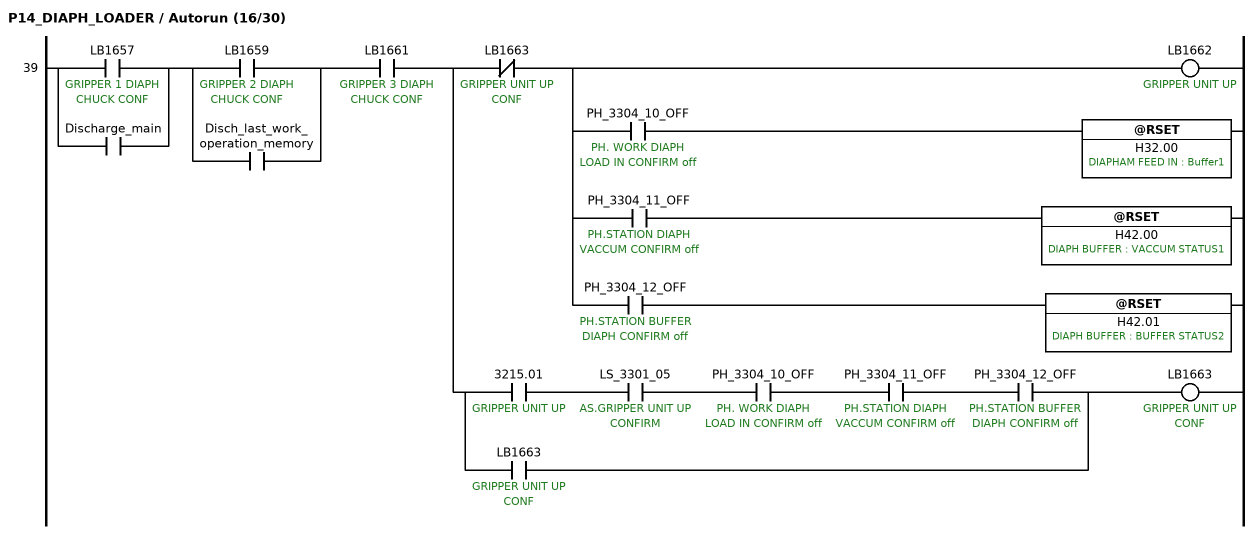
; [picture p192: P14_DIAPH_LOADER / Autorun, rungs 39-39]
; rung 39
LD LB1657  ; GRIPPER 1 DIAPH CHUCK CONF
OR Discharge_main
LD LB1659  ; GRIPPER 2 DIAPH CHUCK CONF
OR Disch_last_work_operation_memory
ANDLD
AND LB1661  ; GRIPPER 3 DIAPH CHUCK CONF
OUT TR0
ANDNOT LB1663  ; GRIPPER UNIT UP CONF
OUT TR1
OUT LB1662  ; GRIPPER UNIT UP
AND PH_3304_10_OFF  ; PH. WORK DIAPH LOAD IN CONFIRM off
@RSET H32.00  ; DIAPHAM FEED IN : Buffer1
LD TR1
AND PH_3304_11_OFF  ; PH.STATION DIAPH VACCUM CONFIRM off
@RSET H42.00  ; DIAPH BUFFER : VACCUM STATUS1
LD TR1
AND PH_3304_12_OFF  ; PH.STATION BUFFER DIAPH CONFIRM off
@RSET H42.01  ; DIAPH BUFFER : BUFFER STATUS2
LD TR0
LD 3215.01  ; GRIPPER UNIT UP
AND LS_3301_05  ; AS.GRIPPER UNIT UP CONFIRM
AND PH_3304_10_OFF  ; PH. WORK DIAPH LOAD IN CONFIRM off
AND PH_3304_11_OFF  ; PH.STATION DIAPH VACCUM CONFIRM off
AND PH_3304_12_OFF  ; PH.STATION BUFFER DIAPH CONFIRM off
OR LB1663  ; GRIPPER UNIT UP CONF
ANDLD
OUT LB1663  ; GRIPPER UNIT UP CONF

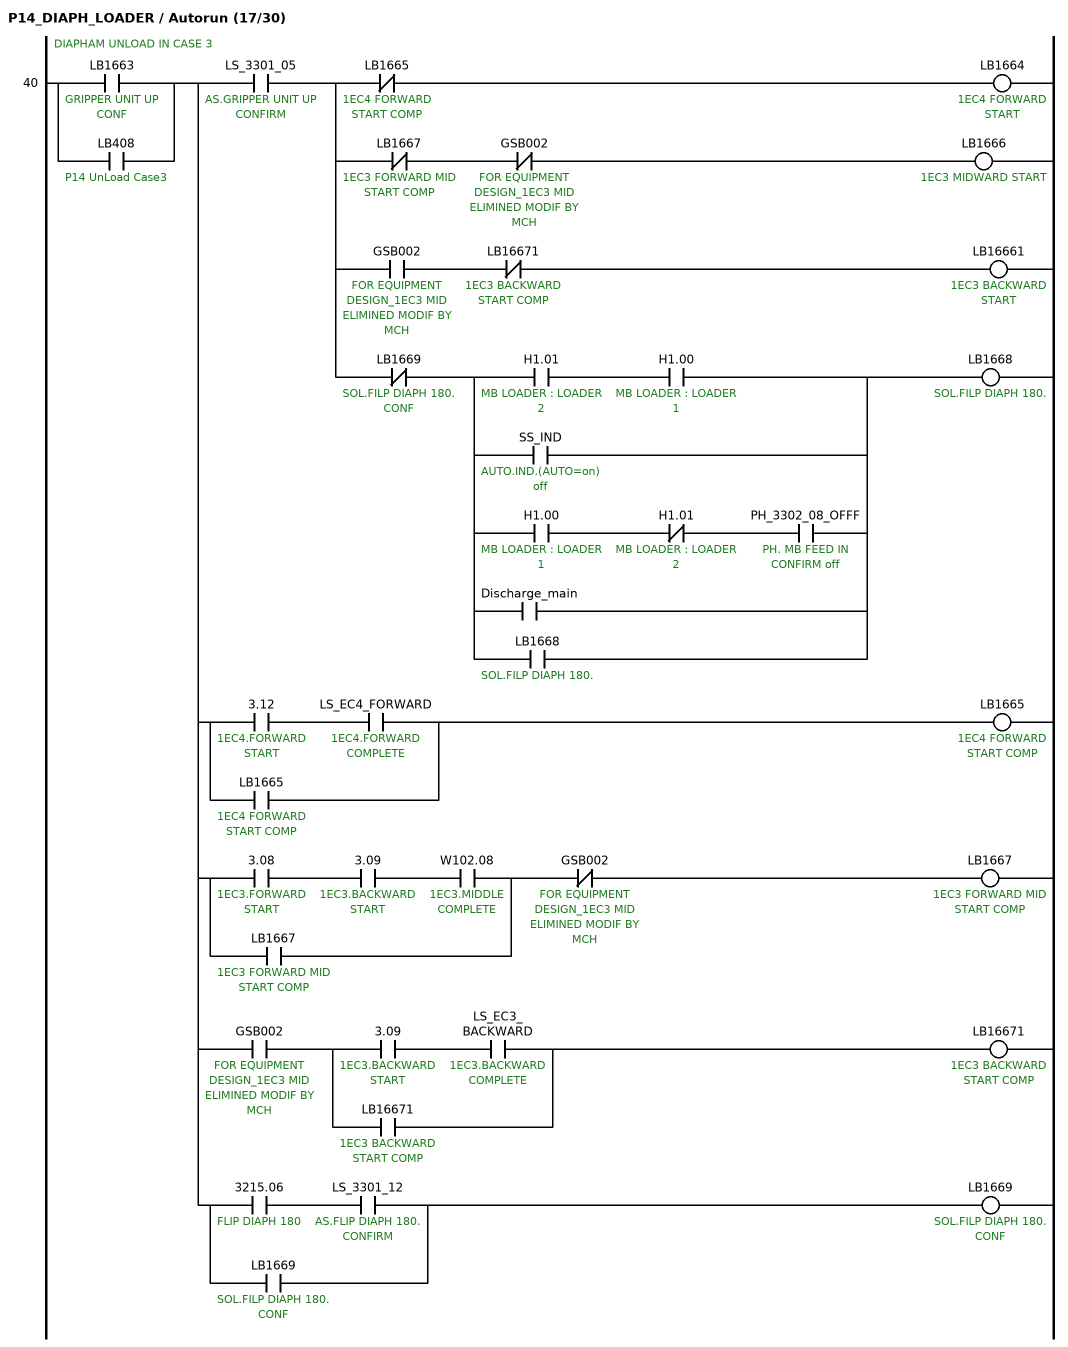
; rung 40: DIAPHAM UNLOAD IN CASE 3
LD LB1663  ; GRIPPER UNIT UP CONF
OR LB408  ; P14 UnLoad Case3
OUT TR0
AND LS_3301_05  ; AS.GRIPPER UNIT UP CONFIRM
OUT TR1
ANDNOT LB1665  ; 1EC4 FORWARD START COMP
OUT LB1664  ; 1EC4 FORWARD START
LD TR1
ANDNOT LB1667  ; 1EC3 FORWARD MID START COMP
ANDNOT GSB002  ; FOR EQUIPMENT DESIGN_1EC3 MID ELIMINED MODIF BY MCH
OUT LB1666  ; 1EC3 MIDWARD START
LD TR1
AND GSB002  ; FOR EQUIPMENT DESIGN_1EC3 MID ELIMINED MODIF BY MCH
ANDNOT LB16671  ; 1EC3 BACKWARD START COMP
OUT LB16661  ; 1EC3 BACKWARD START
LD TR1
ANDNOT LB1669  ; SOL.FILP DIAPH 180. CONF
LD H1.01  ; MB LOADER : LOADER 2
AND H1.00  ; MB LOADER : LOADER 1
OR SS_IND  ; AUTO.IND.(AUTO=on) off
LD H1.00  ; MB LOADER : LOADER 1
ANDNOT H1.01  ; MB LOADER : LOADER 2
AND PH_3302_08_OFFF  ; PH. MB FEED IN CONFIRM off
ORLD
OR Discharge_main
OR LB1668  ; SOL.FILP DIAPH 180.
ANDLD
OUT LB1668  ; SOL.FILP DIAPH 180.
LD TR0
LD 3.12  ; 1EC4.FORWARD START
AND LS_EC4_FORWARD  ; 1EC4.FORWARD COMPLETE
OR LB1665  ; 1EC4 FORWARD START COMP
ANDLD
OUT LB1665  ; 1EC4 FORWARD START COMP
LD TR0
LD 3.08  ; 1EC3.FORWARD START
AND 3.09  ; 1EC3.BACKWARD START
AND W102.08  ; 1EC3.MIDDLE COMPLETE
OR LB1667  ; 1EC3 FORWARD MID START COMP
ANDLD
ANDNOT GSB002  ; FOR EQUIPMENT DESIGN_1EC3 MID ELIMINED MODIF BY MCH
OUT LB1667  ; 1EC3 FORWARD MID START COMP
LD TR0
AND GSB002  ; FOR EQUIPMENT DESIGN_1EC3 MID ELIMINED MODIF BY MCH
LD 3.09  ; 1EC3.BACKWARD START
AND LS_EC3_BACKWARD  ; 1EC3.BACKWARD COMPLETE
OR LB16671  ; 1EC3 BACKWARD START COMP
ANDLD
OUT LB16671  ; 1EC3 BACKWARD START COMP
LD TR0
LD 3215.06  ; FLIP DIAPH 180
AND LS_3301_12  ; AS.FLIP DIAPH 180. CONFIRM
OR LB1669  ; SOL.FILP DIAPH 180. CONF
ANDLD
OUT LB1669  ; SOL.FILP DIAPH 180. CONF

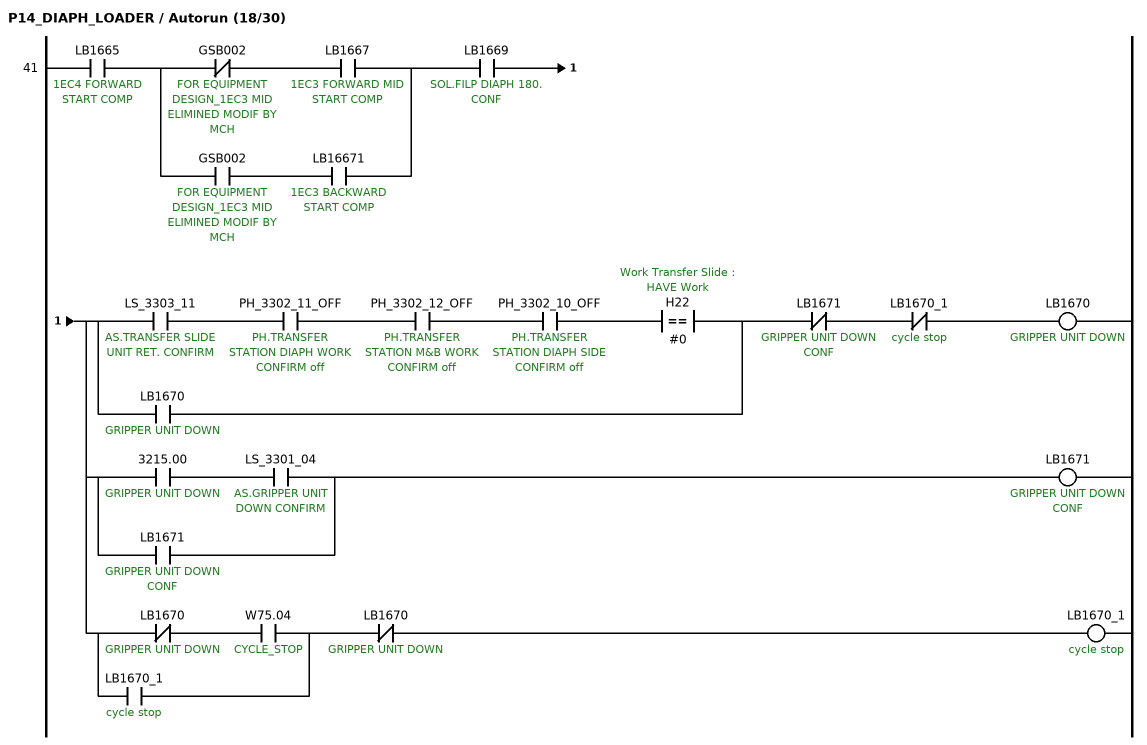
; rung 41
LD LB1665  ; 1EC4 FORWARD START COMP
LDNOT GSB002  ; FOR EQUIPMENT DESIGN_1EC3 MID ELIMINED MODIF BY MCH
AND LB1667  ; 1EC3 FORWARD MID START COMP
LD GSB002  ; FOR EQUIPMENT DESIGN_1EC3 MID ELIMINED MODIF BY MCH
AND LB16671  ; 1EC3 BACKWARD START COMP
ORLD
ANDLD
AND LB1669  ; SOL.FILP DIAPH 180. CONF
OUT TR0
LD LS_3303_11  ; AS.TRANSFER SLIDE UNIT RET. CONFIRM
AND PH_3302_11_OFF  ; PH.TRANSFER STATION DIAPH WORK CONFIRM off
AND PH_3302_12_OFF  ; PH.TRANSFER STATION M&B WORK CONFIRM off
AND PH_3302_10_OFF  ; PH.TRANSFER STATION DIAPH SIDE CONFIRM off
AND=(300) H22 #0  ; Work Transfer Slide : HAVE Work
OR LB1670  ; GRIPPER UNIT DOWN
ANDLD
ANDNOT LB1671  ; GRIPPER UNIT DOWN CONF
ANDNOT LB1670_1  ; cycle stop
OUT LB1670  ; GRIPPER UNIT DOWN
LD TR0
LD 3215.00  ; GRIPPER UNIT DOWN
AND LS_3301_04  ; AS.GRIPPER UNIT DOWN CONFIRM
OR LB1671  ; GRIPPER UNIT DOWN CONF
ANDLD
OUT LB1671  ; GRIPPER UNIT DOWN CONF
LD TR0
LDNOT LB1670  ; GRIPPER UNIT DOWN
AND W75.04  ; CYCLE_STOP
OR LB1670_1  ; cycle stop
ANDLD
ANDNOT LB1670  ; GRIPPER UNIT DOWN
OUT LB1670_1  ; cycle stop

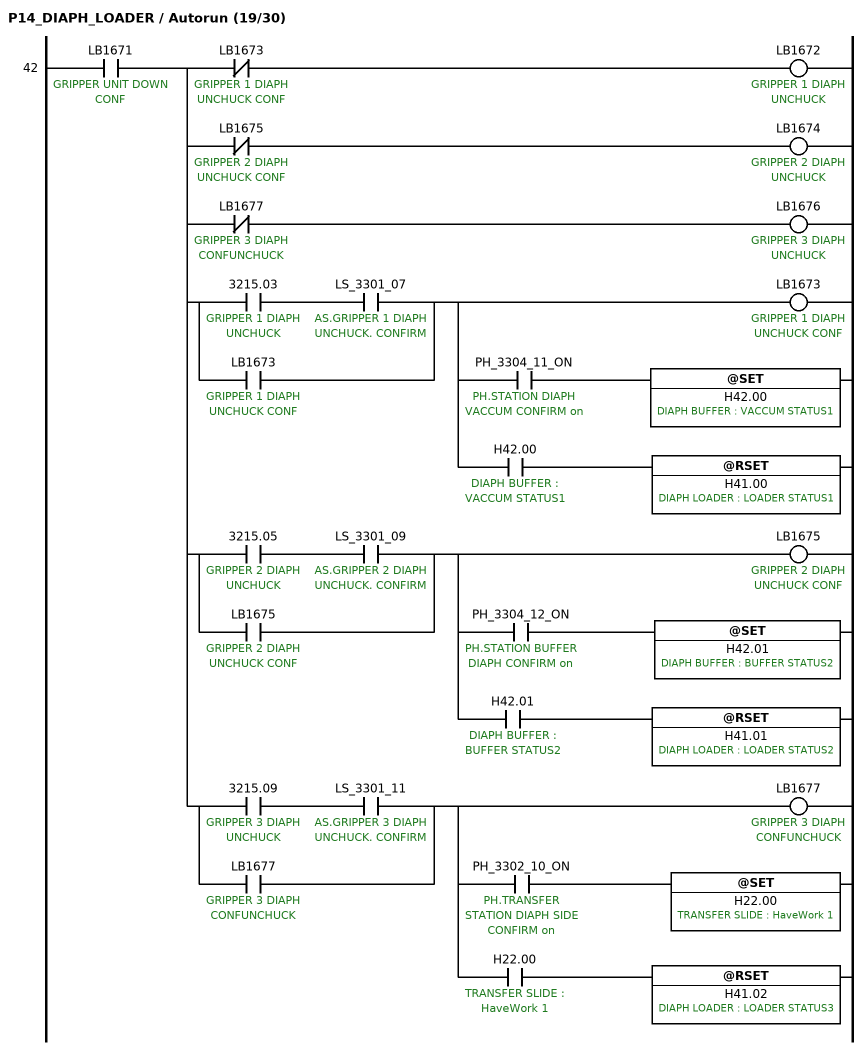
; rung 42
LD LB1671  ; GRIPPER UNIT DOWN CONF
OUT TR0
ANDNOT LB1673  ; GRIPPER 1 DIAPH UNCHUCK CONF
OUT LB1672  ; GRIPPER 1 DIAPH UNCHUCK
LD TR0
ANDNOT LB1675  ; GRIPPER 2 DIAPH UNCHUCK CONF
OUT LB1674  ; GRIPPER 2 DIAPH UNCHUCK
LD TR0
ANDNOT LB1677  ; GRIPPER 3 DIAPH CONFUNCHUCK
OUT LB1676  ; GRIPPER 3 DIAPH UNCHUCK
LD TR0
LD 3215.03  ; GRIPPER 1 DIAPH UNCHUCK
AND LS_3301_07  ; AS.GRIPPER 1 DIAPH UNCHUCK. CONFIRM
OR LB1673  ; GRIPPER 1 DIAPH UNCHUCK CONF
ANDLD
OUT TR1
OUT LB1673  ; GRIPPER 1 DIAPH UNCHUCK CONF
AND PH_3304_11_ON  ; PH.STATION DIAPH VACCUM CONFIRM on
@SET H42.00  ; DIAPH BUFFER : VACCUM STATUS1
LD TR1
AND H42.00  ; DIAPH BUFFER : VACCUM STATUS1
@RSET H41.00  ; DIAPH LOADER : LOADER STATUS1
LD TR0
LD 3215.05  ; GRIPPER 2 DIAPH UNCHUCK
AND LS_3301_09  ; AS.GRIPPER 2 DIAPH UNCHUCK. CONFIRM
OR LB1675  ; GRIPPER 2 DIAPH UNCHUCK CONF
ANDLD
OUT TR1
OUT LB1675  ; GRIPPER 2 DIAPH UNCHUCK CONF
AND PH_3304_12_ON  ; PH.STATION BUFFER DIAPH CONFIRM on
@SET H42.01  ; DIAPH BUFFER : BUFFER STATUS2
LD TR1
AND H42.01  ; DIAPH BUFFER : BUFFER STATUS2
@RSET H41.01  ; DIAPH LOADER : LOADER STATUS2
LD TR0
LD 3215.09  ; GRIPPER 3 DIAPH UNCHUCK
AND LS_3301_11  ; AS.GRIPPER 3 DIAPH UNCHUCK. CONFIRM
OR LB1677  ; GRIPPER 3 DIAPH CONFUNCHUCK
ANDLD
OUT TR0
OUT LB1677  ; GRIPPER 3 DIAPH CONFUNCHUCK
AND PH_3302_10_ON  ; PH.TRANSFER STATION DIAPH SIDE CONFIRM on
@SET H22.00  ; TRANSFER SLIDE : HaveWork 1
LD TR0
AND H22.00  ; TRANSFER SLIDE : HaveWork 1
@RSET H41.02  ; DIAPH LOADER : LOADER STATUS3

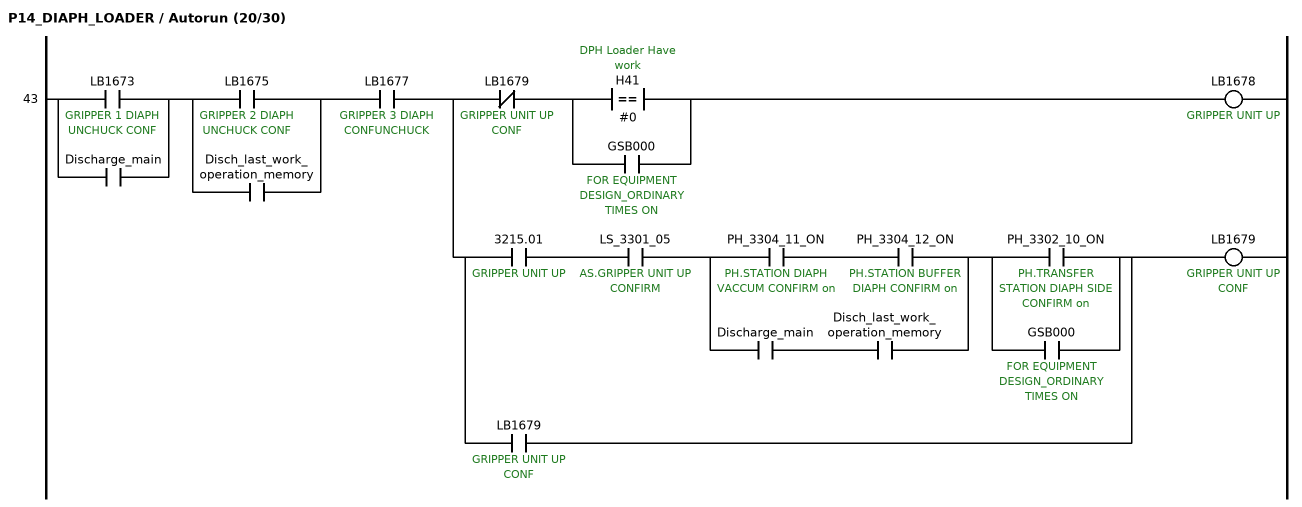
; rung 43
LD LB1673  ; GRIPPER 1 DIAPH UNCHUCK CONF
OR Discharge_main
LD LB1675  ; GRIPPER 2 DIAPH UNCHUCK CONF
OR Disch_last_work_operation_memory
ANDLD
AND LB1677  ; GRIPPER 3 DIAPH CONFUNCHUCK
OUT TR0
ANDNOT LB1679  ; GRIPPER UNIT UP CONF
LD=(300) H41 #0  ; DPH Loader Have work
OR GSB000  ; FOR EQUIPMENT DESIGN_ORDINARY TIMES ON
ANDLD
OUT LB1678  ; GRIPPER UNIT UP
LD TR0
LD 3215.01  ; GRIPPER UNIT UP
AND LS_3301_05  ; AS.GRIPPER UNIT UP CONFIRM
LD PH_3304_11_ON  ; PH.STATION DIAPH VACCUM CONFIRM on
AND PH_3304_12_ON  ; PH.STATION BUFFER DIAPH CONFIRM on
LD Discharge_main
AND Disch_last_work_operation_memory
ORLD
ANDLD
LD PH_3302_10_ON  ; PH.TRANSFER STATION DIAPH SIDE CONFIRM on
OR GSB000  ; FOR EQUIPMENT DESIGN_ORDINARY TIMES ON
ANDLD
OR LB1679  ; GRIPPER UNIT UP CONF
ANDLD
OUT LB1679  ; GRIPPER UNIT UP CONF

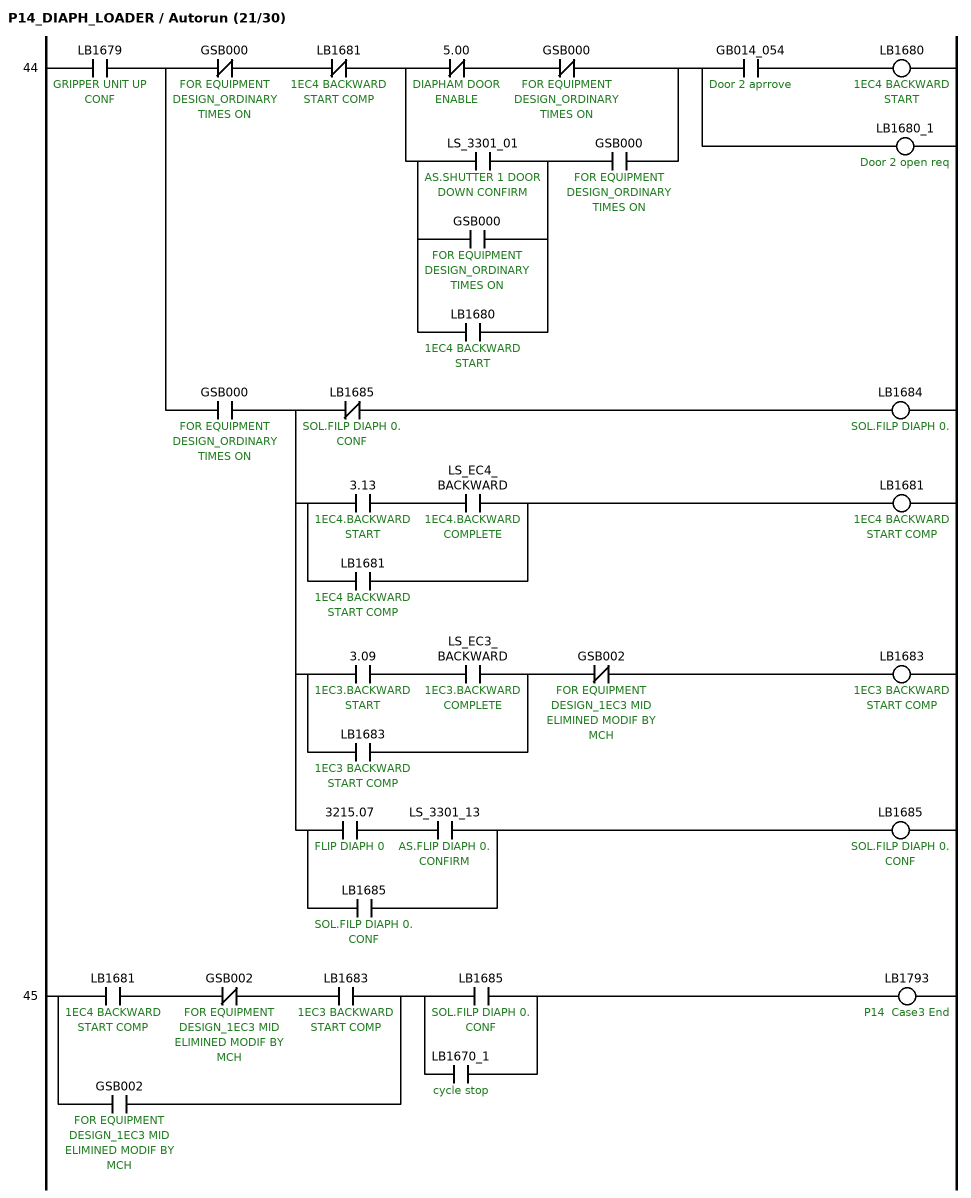
; rung 44
LD LB1679  ; GRIPPER UNIT UP CONF
OUT TR0
ANDNOT GSB000  ; FOR EQUIPMENT DESIGN_ORDINARY TIMES ON
ANDNOT LB1681  ; 1EC4 BACKWARD START COMP
LDNOT 5.00  ; DIAPHAM DOOR ENABLE
ANDNOT GSB000  ; FOR EQUIPMENT DESIGN_ORDINARY TIMES ON
LD LS_3301_01  ; AS.SHUTTER 1 DOOR DOWN CONFIRM
OR GSB000  ; FOR EQUIPMENT DESIGN_ORDINARY TIMES ON
OR LB1680  ; 1EC4 BACKWARD START
AND GSB000  ; FOR EQUIPMENT DESIGN_ORDINARY TIMES ON
ORLD
ANDLD
OUT TR1
AND GB014_054  ; Door 2 aprrove
OUT LB1680  ; 1EC4 BACKWARD START
LD TR1
OUT LB1680_1  ; Door 2 open req
LD TR0
AND GSB000  ; FOR EQUIPMENT DESIGN_ORDINARY TIMES ON
OUT TR0
ANDNOT LB1685  ; SOL.FILP DIAPH 0. CONF
OUT LB1684  ; SOL.FILP DIAPH 0.
LD TR0
LD 3.13  ; 1EC4.BACKWARD START
AND LS_EC4_BACKWARD  ; 1EC4.BACKWARD COMPLETE
OR LB1681  ; 1EC4 BACKWARD START COMP
ANDLD
OUT LB1681  ; 1EC4 BACKWARD START COMP
LD TR0
LD 3.09  ; 1EC3.BACKWARD START
AND LS_EC3_BACKWARD  ; 1EC3.BACKWARD COMPLETE
OR LB1683  ; 1EC3 BACKWARD START COMP
ANDLD
ANDNOT GSB002  ; FOR EQUIPMENT DESIGN_1EC3 MID ELIMINED MODIF BY MCH
OUT LB1683  ; 1EC3 BACKWARD START COMP
LD TR0
LD 3215.07  ; FLIP DIAPH 0
AND LS_3301_13  ; AS.FLIP DIAPH 0. CONFIRM
OR LB1685  ; SOL.FILP DIAPH 0. CONF
ANDLD
OUT LB1685  ; SOL.FILP DIAPH 0. CONF
; rung 45
LD LB1681  ; 1EC4 BACKWARD START COMP
ANDNOT GSB002  ; FOR EQUIPMENT DESIGN_1EC3 MID ELIMINED MODIF BY MCH
AND LB1683  ; 1EC3 BACKWARD START COMP
OR GSB002  ; FOR EQUIPMENT DESIGN_1EC3 MID ELIMINED MODIF BY MCH
LD LB1685  ; SOL.FILP DIAPH 0. CONF
OR LB1670_1  ; cycle stop
ANDLD
OUT LB1793  ; P14  Case3 End

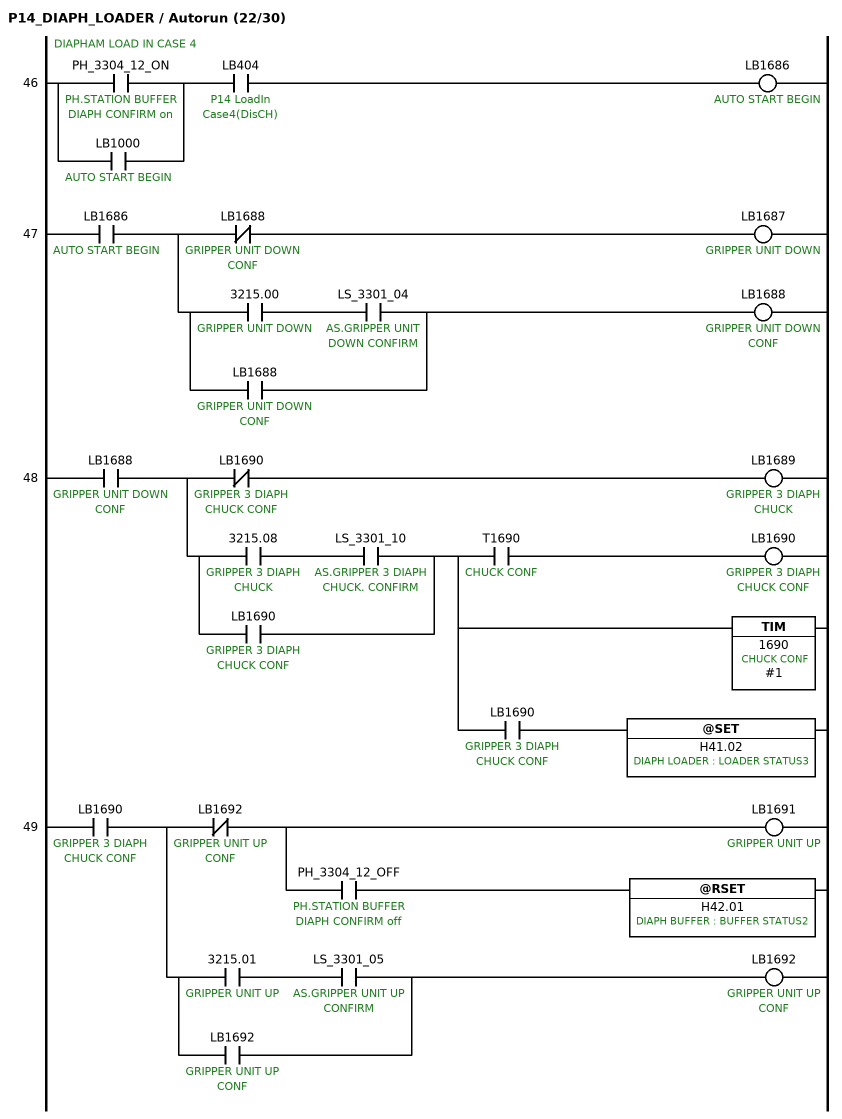
; rung 46: DIAPHAM LOAD IN CASE 4
LD PH_3304_12_ON  ; PH.STATION BUFFER DIAPH CONFIRM on
OR LB1000  ; AUTO START BEGIN
AND LB404  ; P14 LoadIn Case4(DisCH)
OUT LB1686  ; AUTO START BEGIN
; rung 47
LD LB1686  ; AUTO START BEGIN
OUT TR0
ANDNOT LB1688  ; GRIPPER UNIT DOWN CONF
OUT LB1687  ; GRIPPER UNIT DOWN
LD TR0
LD 3215.00  ; GRIPPER UNIT DOWN
AND LS_3301_04  ; AS.GRIPPER UNIT DOWN CONFIRM
OR LB1688  ; GRIPPER UNIT DOWN CONF
ANDLD
OUT LB1688  ; GRIPPER UNIT DOWN CONF
; rung 48
LD LB1688  ; GRIPPER UNIT DOWN CONF
OUT TR0
ANDNOT LB1690  ; GRIPPER 3 DIAPH CHUCK CONF
OUT LB1689  ; GRIPPER 3 DIAPH CHUCK
LD TR0
LD 3215.08  ; GRIPPER 3 DIAPH CHUCK
AND LS_3301_10  ; AS.GRIPPER 3 DIAPH CHUCK. CONFIRM
OR LB1690  ; GRIPPER 3 DIAPH CHUCK CONF
ANDLD
OUT TR0
AND T1690  ; CHUCK CONF
OUT LB1690  ; GRIPPER 3 DIAPH CHUCK CONF
LD TR0
TIM 1690 #1  ; CHUCK CONF
AND LB1690  ; GRIPPER 3 DIAPH CHUCK CONF
@SET H41.02  ; DIAPH LOADER : LOADER STATUS3
; rung 49
LD LB1690  ; GRIPPER 3 DIAPH CHUCK CONF
OUT TR0
ANDNOT LB1692  ; GRIPPER UNIT UP CONF
OUT LB1691  ; GRIPPER UNIT UP
AND PH_3304_12_OFF  ; PH.STATION BUFFER DIAPH CONFIRM off
@RSET H42.01  ; DIAPH BUFFER : BUFFER STATUS2
LD TR0
LD 3215.01  ; GRIPPER UNIT UP
AND LS_3301_05  ; AS.GRIPPER UNIT UP CONFIRM
OR LB1692  ; GRIPPER UNIT UP CONF
ANDLD
OUT LB1692  ; GRIPPER UNIT UP CONF

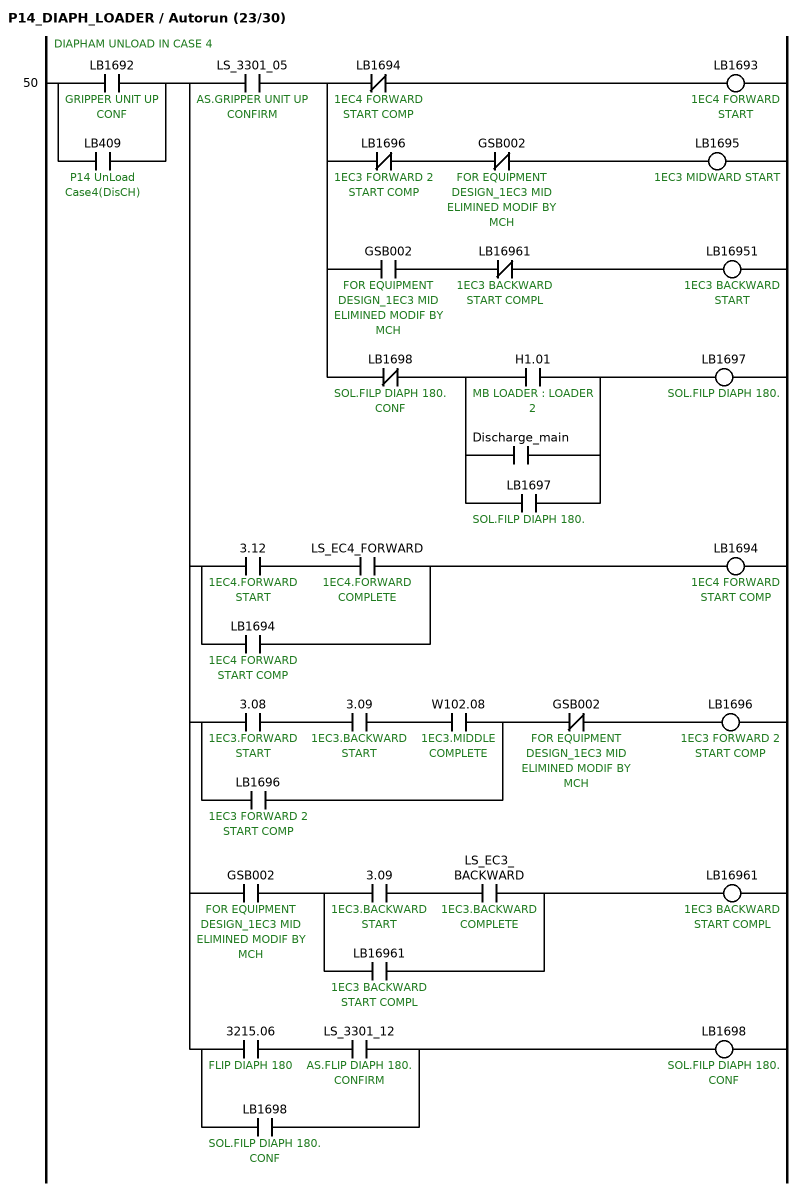
; rung 50: DIAPHAM UNLOAD IN CASE 4
LD LB1692  ; GRIPPER UNIT UP CONF
OR LB409  ; P14 UnLoad Case4(DisCH)
OUT TR0
AND LS_3301_05  ; AS.GRIPPER UNIT UP CONFIRM
OUT TR1
ANDNOT LB1694  ; 1EC4 FORWARD START COMP
OUT LB1693  ; 1EC4 FORWARD START
LD TR1
ANDNOT LB1696  ; 1EC3 FORWARD 2 START COMP
ANDNOT GSB002  ; FOR EQUIPMENT DESIGN_1EC3 MID ELIMINED MODIF BY MCH
OUT LB1695  ; 1EC3 MIDWARD START
LD TR1
AND GSB002  ; FOR EQUIPMENT DESIGN_1EC3 MID ELIMINED MODIF BY MCH
ANDNOT LB16961  ; 1EC3 BACKWARD START COMPL
OUT LB16951  ; 1EC3 BACKWARD START
LD TR1
ANDNOT LB1698  ; SOL.FILP DIAPH 180. CONF
LD H1.01  ; MB LOADER : LOADER 2
OR Discharge_main
OR LB1697  ; SOL.FILP DIAPH 180.
ANDLD
OUT LB1697  ; SOL.FILP DIAPH 180.
LD TR0
LD 3.12  ; 1EC4.FORWARD START
AND LS_EC4_FORWARD  ; 1EC4.FORWARD COMPLETE
OR LB1694  ; 1EC4 FORWARD START COMP
ANDLD
OUT LB1694  ; 1EC4 FORWARD START COMP
LD TR0
LD 3.08  ; 1EC3.FORWARD START
AND 3.09  ; 1EC3.BACKWARD START
AND W102.08  ; 1EC3.MIDDLE COMPLETE
OR LB1696  ; 1EC3 FORWARD 2 START COMP
ANDLD
ANDNOT GSB002  ; FOR EQUIPMENT DESIGN_1EC3 MID ELIMINED MODIF BY MCH
OUT LB1696  ; 1EC3 FORWARD 2 START COMP
LD TR0
AND GSB002  ; FOR EQUIPMENT DESIGN_1EC3 MID ELIMINED MODIF BY MCH
LD 3.09  ; 1EC3.BACKWARD START
AND LS_EC3_BACKWARD  ; 1EC3.BACKWARD COMPLETE
OR LB16961  ; 1EC3 BACKWARD START COMPL
ANDLD
OUT LB16961  ; 1EC3 BACKWARD START COMPL
LD TR0
LD 3215.06  ; FLIP DIAPH 180
AND LS_3301_12  ; AS.FLIP DIAPH 180. CONFIRM
OR LB1698  ; SOL.FILP DIAPH 180. CONF
ANDLD
OUT LB1698  ; SOL.FILP DIAPH 180. CONF

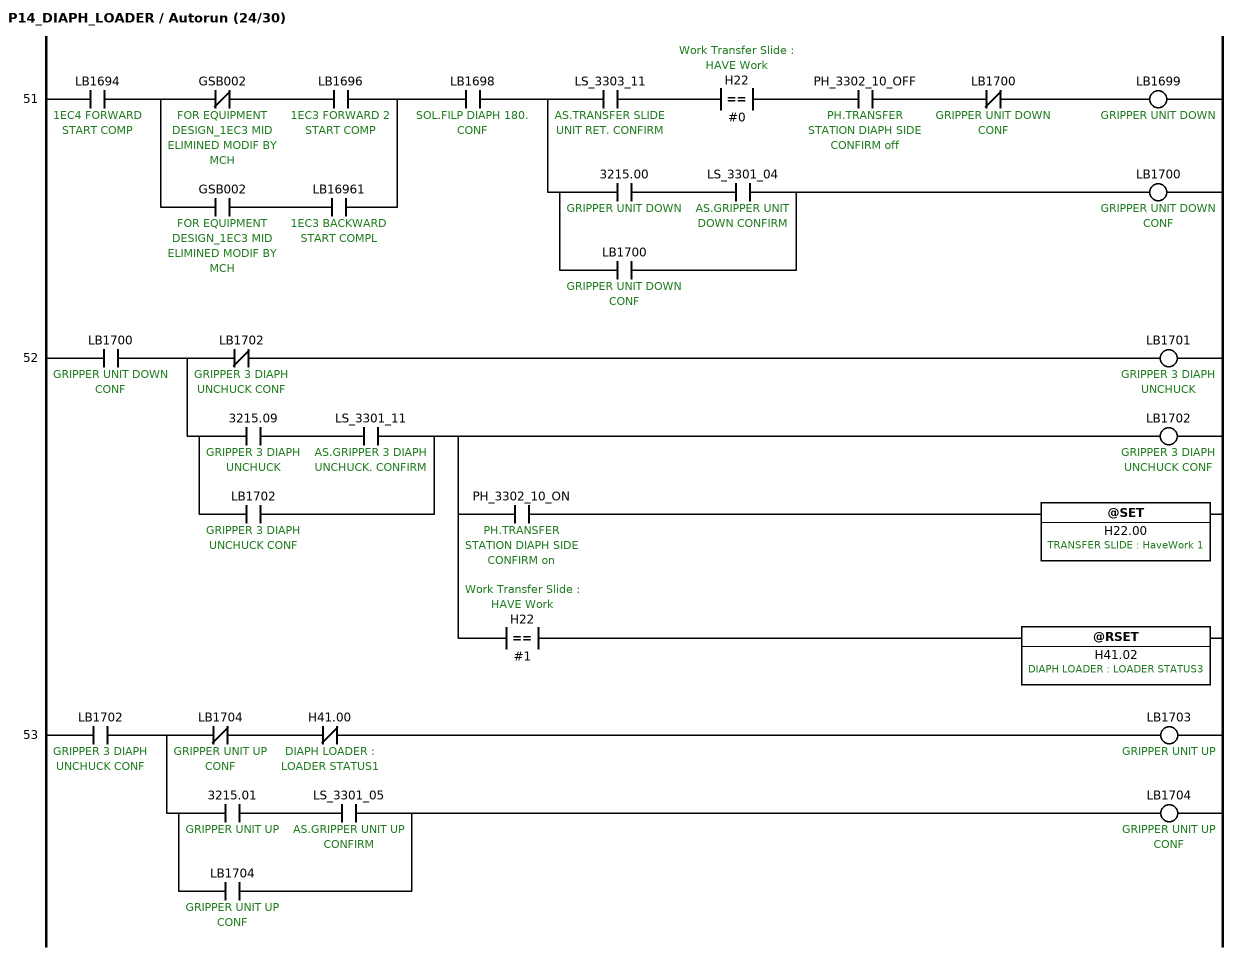
; rung 51
LD LB1694  ; 1EC4 FORWARD START COMP
LDNOT GSB002  ; FOR EQUIPMENT DESIGN_1EC3 MID ELIMINED MODIF BY MCH
AND LB1696  ; 1EC3 FORWARD 2 START COMP
LD GSB002  ; FOR EQUIPMENT DESIGN_1EC3 MID ELIMINED MODIF BY MCH
AND LB16961  ; 1EC3 BACKWARD START COMPL
ORLD
ANDLD
AND LB1698  ; SOL.FILP DIAPH 180. CONF
OUT TR0
AND LS_3303_11  ; AS.TRANSFER SLIDE UNIT RET. CONFIRM
AND=(300) H22 #0  ; Work Transfer Slide : HAVE Work
AND PH_3302_10_OFF  ; PH.TRANSFER STATION DIAPH SIDE CONFIRM off
ANDNOT LB1700  ; GRIPPER UNIT DOWN CONF
OUT LB1699  ; GRIPPER UNIT DOWN
LD TR0
LD 3215.00  ; GRIPPER UNIT DOWN
AND LS_3301_04  ; AS.GRIPPER UNIT DOWN CONFIRM
OR LB1700  ; GRIPPER UNIT DOWN CONF
ANDLD
OUT LB1700  ; GRIPPER UNIT DOWN CONF
; rung 52
LD LB1700  ; GRIPPER UNIT DOWN CONF
OUT TR0
ANDNOT LB1702  ; GRIPPER 3 DIAPH UNCHUCK CONF
OUT LB1701  ; GRIPPER 3 DIAPH UNCHUCK
LD TR0
LD 3215.09  ; GRIPPER 3 DIAPH UNCHUCK
AND LS_3301_11  ; AS.GRIPPER 3 DIAPH UNCHUCK. CONFIRM
OR LB1702  ; GRIPPER 3 DIAPH UNCHUCK CONF
ANDLD
OUT TR0
OUT LB1702  ; GRIPPER 3 DIAPH UNCHUCK CONF
AND PH_3302_10_ON  ; PH.TRANSFER STATION DIAPH SIDE CONFIRM on
@SET H22.00  ; TRANSFER SLIDE : HaveWork 1
LD TR0
AND=(300) H22 #1  ; Work Transfer Slide : HAVE Work
@RSET H41.02  ; DIAPH LOADER : LOADER STATUS3
; rung 53
LD LB1702  ; GRIPPER 3 DIAPH UNCHUCK CONF
OUT TR0
ANDNOT LB1704  ; GRIPPER UNIT UP CONF
ANDNOT H41.00  ; DIAPH LOADER : LOADER STATUS1
OUT LB1703  ; GRIPPER UNIT UP
LD TR0
LD 3215.01  ; GRIPPER UNIT UP
AND LS_3301_05  ; AS.GRIPPER UNIT UP CONFIRM
OR LB1704  ; GRIPPER UNIT UP CONF
ANDLD
OUT LB1704  ; GRIPPER UNIT UP CONF

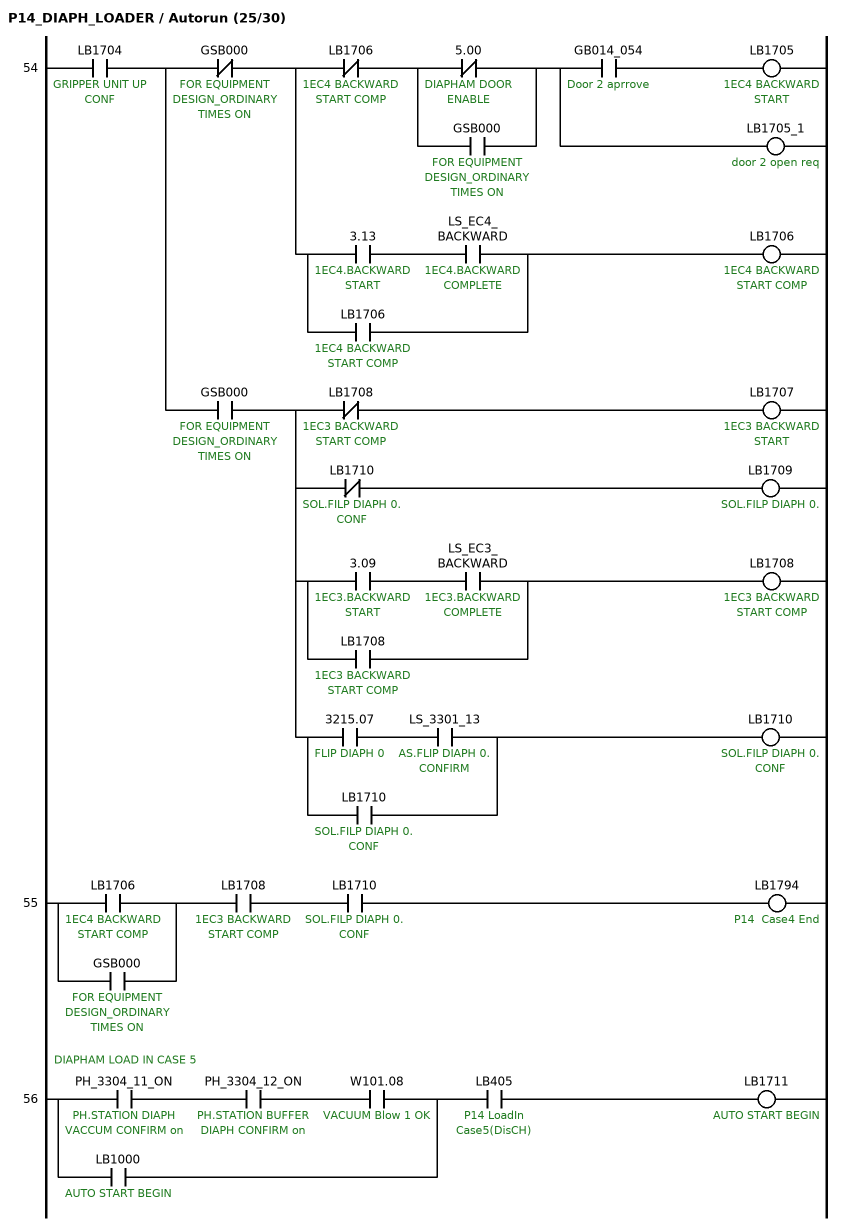
; rung 54
LD LB1704  ; GRIPPER UNIT UP CONF
OUT TR0
ANDNOT GSB000  ; FOR EQUIPMENT DESIGN_ORDINARY TIMES ON
OUT TR1
ANDNOT LB1706  ; 1EC4 BACKWARD START COMP
LDNOT 5.00  ; DIAPHAM DOOR ENABLE
OR GSB000  ; FOR EQUIPMENT DESIGN_ORDINARY TIMES ON
ANDLD
OUT TR2
AND GB014_054  ; Door 2 aprrove
OUT LB1705  ; 1EC4 BACKWARD START
LD TR2
OUT LB1705_1  ; door 2 open req
LD TR1
LD 3.13  ; 1EC4.BACKWARD START
AND LS_EC4_BACKWARD  ; 1EC4.BACKWARD COMPLETE
OR LB1706  ; 1EC4 BACKWARD START COMP
ANDLD
OUT LB1706  ; 1EC4 BACKWARD START COMP
LD TR0
AND GSB000  ; FOR EQUIPMENT DESIGN_ORDINARY TIMES ON
OUT TR0
ANDNOT LB1708  ; 1EC3 BACKWARD START COMP
OUT LB1707  ; 1EC3 BACKWARD START
LD TR0
ANDNOT LB1710  ; SOL.FILP DIAPH 0. CONF
OUT LB1709  ; SOL.FILP DIAPH 0.
LD TR0
LD 3.09  ; 1EC3.BACKWARD START
AND LS_EC3_BACKWARD  ; 1EC3.BACKWARD COMPLETE
OR LB1708  ; 1EC3 BACKWARD START COMP
ANDLD
OUT LB1708  ; 1EC3 BACKWARD START COMP
LD TR0
LD 3215.07  ; FLIP DIAPH 0
AND LS_3301_13  ; AS.FLIP DIAPH 0. CONFIRM
OR LB1710  ; SOL.FILP DIAPH 0. CONF
ANDLD
OUT LB1710  ; SOL.FILP DIAPH 0. CONF
; rung 55
LD LB1706  ; 1EC4 BACKWARD START COMP
OR GSB000  ; FOR EQUIPMENT DESIGN_ORDINARY TIMES ON
AND LB1708  ; 1EC3 BACKWARD START COMP
AND LB1710  ; SOL.FILP DIAPH 0. CONF
OUT LB1794  ; P14  Case4 End
; rung 56: DIAPHAM LOAD IN CASE 5
LD PH_3304_11_ON  ; PH.STATION DIAPH VACCUM CONFIRM on
AND PH_3304_12_ON  ; PH.STATION BUFFER DIAPH CONFIRM on
AND W101.08  ; VACUUM Blow 1 OK
OR LB1000  ; AUTO START BEGIN
AND LB405  ; P14 LoadIn Case5(DisCH)
OUT LB1711  ; AUTO START BEGIN

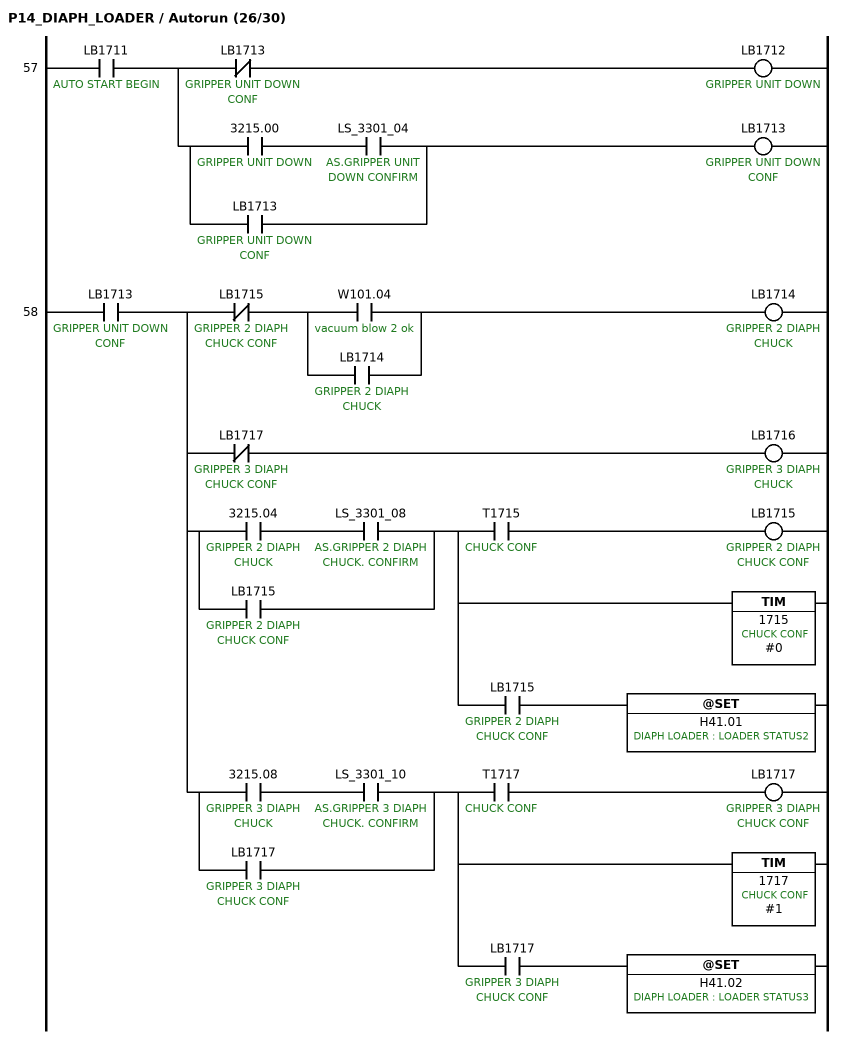
; rung 57
LD LB1711  ; AUTO START BEGIN
OUT TR0
ANDNOT LB1713  ; GRIPPER UNIT DOWN CONF
OUT LB1712  ; GRIPPER UNIT DOWN
LD TR0
LD 3215.00  ; GRIPPER UNIT DOWN
AND LS_3301_04  ; AS.GRIPPER UNIT DOWN CONFIRM
OR LB1713  ; GRIPPER UNIT DOWN CONF
ANDLD
OUT LB1713  ; GRIPPER UNIT DOWN CONF
; rung 58
LD LB1713  ; GRIPPER UNIT DOWN CONF
OUT TR0
ANDNOT LB1715  ; GRIPPER 2 DIAPH CHUCK CONF
LD W101.04  ; vacuum blow 2 ok
OR LB1714  ; GRIPPER 2 DIAPH CHUCK
ANDLD
OUT LB1714  ; GRIPPER 2 DIAPH CHUCK
LD TR0
ANDNOT LB1717  ; GRIPPER 3 DIAPH CHUCK CONF
OUT LB1716  ; GRIPPER 3 DIAPH CHUCK
LD TR0
LD 3215.04  ; GRIPPER 2 DIAPH CHUCK
AND LS_3301_08  ; AS.GRIPPER 2 DIAPH CHUCK. CONFIRM
OR LB1715  ; GRIPPER 2 DIAPH CHUCK CONF
ANDLD
OUT TR1
AND T1715  ; CHUCK CONF
OUT LB1715  ; GRIPPER 2 DIAPH CHUCK CONF
LD TR1
TIM 1715 #0  ; CHUCK CONF
AND LB1715  ; GRIPPER 2 DIAPH CHUCK CONF
@SET H41.01  ; DIAPH LOADER : LOADER STATUS2
LD TR0
LD 3215.08  ; GRIPPER 3 DIAPH CHUCK
AND LS_3301_10  ; AS.GRIPPER 3 DIAPH CHUCK. CONFIRM
OR LB1717  ; GRIPPER 3 DIAPH CHUCK CONF
ANDLD
OUT TR0
AND T1717  ; CHUCK CONF
OUT LB1717  ; GRIPPER 3 DIAPH CHUCK CONF
LD TR0
TIM 1717 #1  ; CHUCK CONF
AND LB1717  ; GRIPPER 3 DIAPH CHUCK CONF
@SET H41.02  ; DIAPH LOADER : LOADER STATUS3

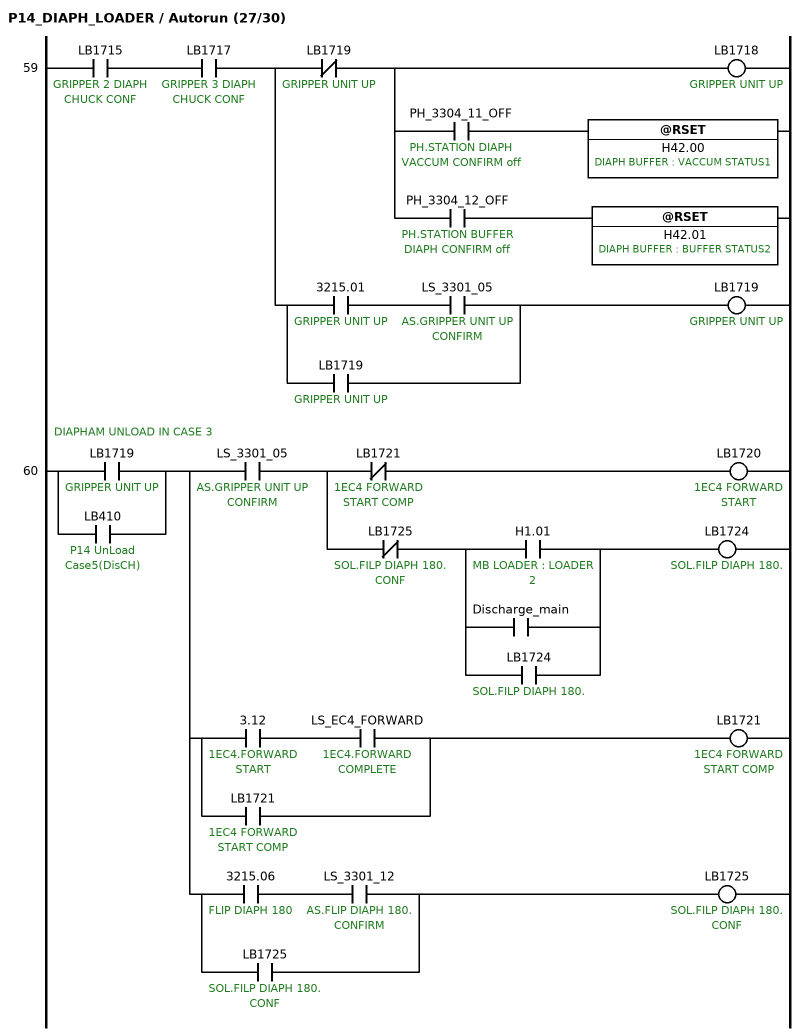
; rung 59
LD LB1715  ; GRIPPER 2 DIAPH CHUCK CONF
AND LB1717  ; GRIPPER 3 DIAPH CHUCK CONF
OUT TR0
ANDNOT LB1719  ; GRIPPER UNIT UP
OUT TR1
OUT LB1718  ; GRIPPER UNIT UP
AND PH_3304_11_OFF  ; PH.STATION DIAPH VACCUM CONFIRM off
@RSET H42.00  ; DIAPH BUFFER : VACCUM STATUS1
LD TR1
AND PH_3304_12_OFF  ; PH.STATION BUFFER DIAPH CONFIRM off
@RSET H42.01  ; DIAPH BUFFER : BUFFER STATUS2
LD TR0
LD 3215.01  ; GRIPPER UNIT UP
AND LS_3301_05  ; AS.GRIPPER UNIT UP CONFIRM
OR LB1719  ; GRIPPER UNIT UP
ANDLD
OUT LB1719  ; GRIPPER UNIT UP
; rung 60: DIAPHAM UNLOAD IN CASE 3
LD LB1719  ; GRIPPER UNIT UP
OR LB410  ; P14 UnLoad Case5(DisCH)
OUT TR0
AND LS_3301_05  ; AS.GRIPPER UNIT UP CONFIRM
OUT TR1
ANDNOT LB1721  ; 1EC4 FORWARD START COMP
OUT LB1720  ; 1EC4 FORWARD START
LD TR1
ANDNOT LB1725  ; SOL.FILP DIAPH 180. CONF
LD H1.01  ; MB LOADER : LOADER 2
OR Discharge_main
OR LB1724  ; SOL.FILP DIAPH 180.
ANDLD
OUT LB1724  ; SOL.FILP DIAPH 180.
LD TR0
LD 3.12  ; 1EC4.FORWARD START
AND LS_EC4_FORWARD  ; 1EC4.FORWARD COMPLETE
OR LB1721  ; 1EC4 FORWARD START COMP
ANDLD
OUT LB1721  ; 1EC4 FORWARD START COMP
LD TR0
LD 3215.06  ; FLIP DIAPH 180
AND LS_3301_12  ; AS.FLIP DIAPH 180. CONFIRM
OR LB1725  ; SOL.FILP DIAPH 180. CONF
ANDLD
OUT LB1725  ; SOL.FILP DIAPH 180. CONF

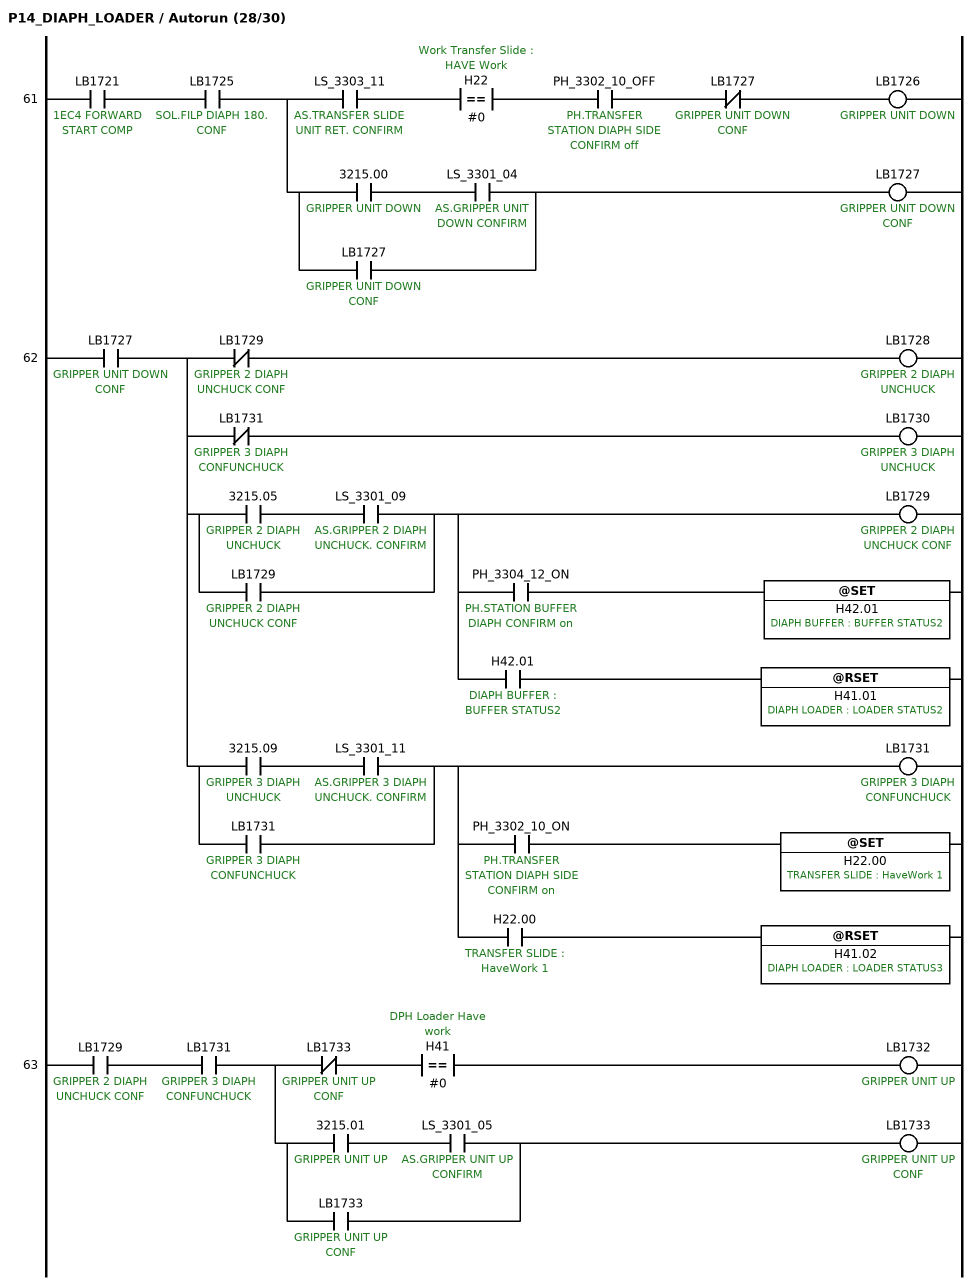
; rung 61
LD LB1721  ; 1EC4 FORWARD START COMP
AND LB1725  ; SOL.FILP DIAPH 180. CONF
OUT TR0
AND LS_3303_11  ; AS.TRANSFER SLIDE UNIT RET. CONFIRM
AND=(300) H22 #0  ; Work Transfer Slide : HAVE Work
AND PH_3302_10_OFF  ; PH.TRANSFER STATION DIAPH SIDE CONFIRM off
ANDNOT LB1727  ; GRIPPER UNIT DOWN CONF
OUT LB1726  ; GRIPPER UNIT DOWN
LD TR0
LD 3215.00  ; GRIPPER UNIT DOWN
AND LS_3301_04  ; AS.GRIPPER UNIT DOWN CONFIRM
OR LB1727  ; GRIPPER UNIT DOWN CONF
ANDLD
OUT LB1727  ; GRIPPER UNIT DOWN CONF
; rung 62
LD LB1727  ; GRIPPER UNIT DOWN CONF
OUT TR0
ANDNOT LB1729  ; GRIPPER 2 DIAPH UNCHUCK CONF
OUT LB1728  ; GRIPPER 2 DIAPH UNCHUCK
LD TR0
ANDNOT LB1731  ; GRIPPER 3 DIAPH CONFUNCHUCK
OUT LB1730  ; GRIPPER 3 DIAPH UNCHUCK
LD TR0
LD 3215.05  ; GRIPPER 2 DIAPH UNCHUCK
AND LS_3301_09  ; AS.GRIPPER 2 DIAPH UNCHUCK. CONFIRM
OR LB1729  ; GRIPPER 2 DIAPH UNCHUCK CONF
ANDLD
OUT TR1
OUT LB1729  ; GRIPPER 2 DIAPH UNCHUCK CONF
AND PH_3304_12_ON  ; PH.STATION BUFFER DIAPH CONFIRM on
@SET H42.01  ; DIAPH BUFFER : BUFFER STATUS2
LD TR1
AND H42.01  ; DIAPH BUFFER : BUFFER STATUS2
@RSET H41.01  ; DIAPH LOADER : LOADER STATUS2
LD TR0
LD 3215.09  ; GRIPPER 3 DIAPH UNCHUCK
AND LS_3301_11  ; AS.GRIPPER 3 DIAPH UNCHUCK. CONFIRM
OR LB1731  ; GRIPPER 3 DIAPH CONFUNCHUCK
ANDLD
OUT TR0
OUT LB1731  ; GRIPPER 3 DIAPH CONFUNCHUCK
AND PH_3302_10_ON  ; PH.TRANSFER STATION DIAPH SIDE CONFIRM on
@SET H22.00  ; TRANSFER SLIDE : HaveWork 1
LD TR0
AND H22.00  ; TRANSFER SLIDE : HaveWork 1
@RSET H41.02  ; DIAPH LOADER : LOADER STATUS3
; rung 63
LD LB1729  ; GRIPPER 2 DIAPH UNCHUCK CONF
AND LB1731  ; GRIPPER 3 DIAPH CONFUNCHUCK
OUT TR0
ANDNOT LB1733  ; GRIPPER UNIT UP CONF
AND=(300) H41 #0  ; DPH Loader Have work
OUT LB1732  ; GRIPPER UNIT UP
LD TR0
LD 3215.01  ; GRIPPER UNIT UP
AND LS_3301_05  ; AS.GRIPPER UNIT UP CONFIRM
OR LB1733  ; GRIPPER UNIT UP CONF
ANDLD
OUT LB1733  ; GRIPPER UNIT UP CONF

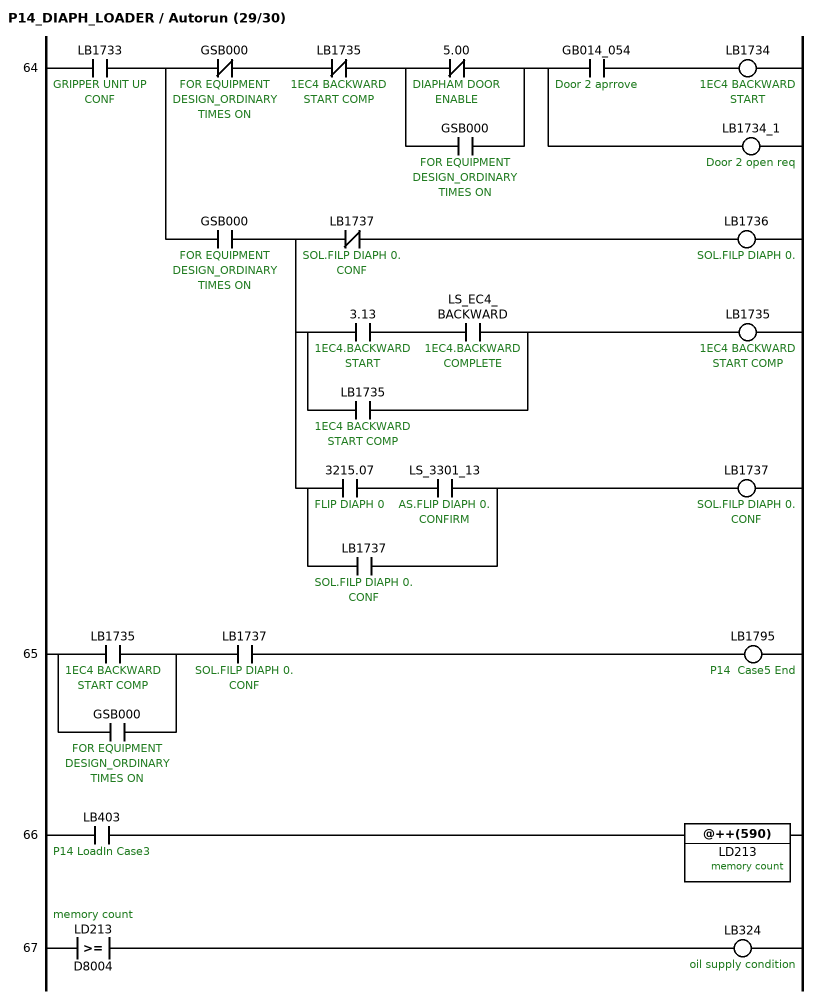
; rung 64
LD LB1733  ; GRIPPER UNIT UP CONF
OUT TR0
ANDNOT GSB000  ; FOR EQUIPMENT DESIGN_ORDINARY TIMES ON
ANDNOT LB1735  ; 1EC4 BACKWARD START COMP
LDNOT 5.00  ; DIAPHAM DOOR ENABLE
OR GSB000  ; FOR EQUIPMENT DESIGN_ORDINARY TIMES ON
ANDLD
OUT TR1
AND GB014_054  ; Door 2 aprrove
OUT LB1734  ; 1EC4 BACKWARD START
LD TR1
OUT LB1734_1  ; Door 2 open req
LD TR0
AND GSB000  ; FOR EQUIPMENT DESIGN_ORDINARY TIMES ON
OUT TR0
ANDNOT LB1737  ; SOL.FILP DIAPH 0. CONF
OUT LB1736  ; SOL.FILP DIAPH 0.
LD TR0
LD 3.13  ; 1EC4.BACKWARD START
AND LS_EC4_BACKWARD  ; 1EC4.BACKWARD COMPLETE
OR LB1735  ; 1EC4 BACKWARD START COMP
ANDLD
OUT LB1735  ; 1EC4 BACKWARD START COMP
LD TR0
LD 3215.07  ; FLIP DIAPH 0
AND LS_3301_13  ; AS.FLIP DIAPH 0. CONFIRM
OR LB1737  ; SOL.FILP DIAPH 0. CONF
ANDLD
OUT LB1737  ; SOL.FILP DIAPH 0. CONF
; rung 65
LD LB1735  ; 1EC4 BACKWARD START COMP
OR GSB000  ; FOR EQUIPMENT DESIGN_ORDINARY TIMES ON
AND LB1737  ; SOL.FILP DIAPH 0. CONF
OUT LB1795  ; P14  Case5 End
; rung 66
LD LB403  ; P14 LoadIn Case3
@++(590) LD213  ; memory count
; rung 67
LD>=(325) LD213 D8004  ; memory count
OUT LB324  ; oil supply condition

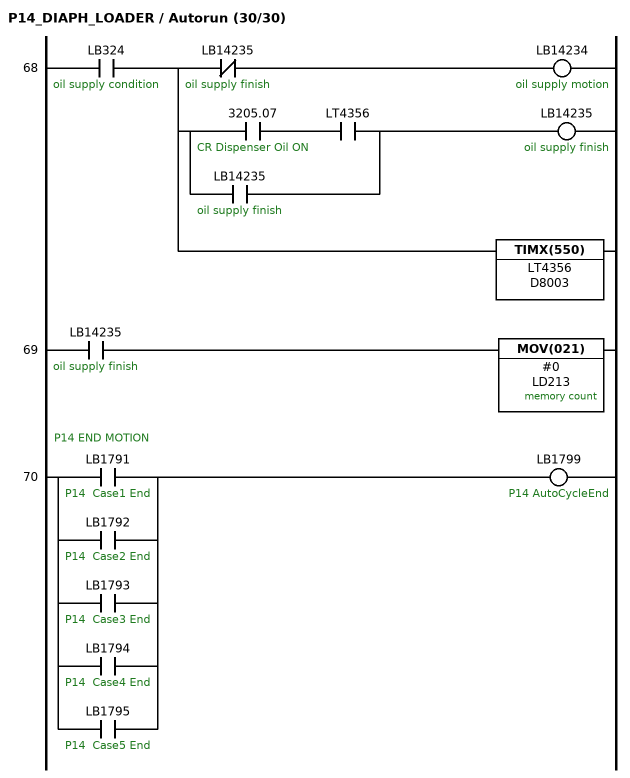
; rung 68
LD LB324  ; oil supply condition
OUT TR0
ANDNOT LB14235  ; oil supply finish
OUT LB14234  ; oil supply motion
LD TR0
LD 3205.07  ; CR Dispenser Oil ON
AND LT4356
OR LB14235  ; oil supply finish
ANDLD
OUT LB14235  ; oil supply finish
LD TR0
TIMX(550) LT4356 D8003
; rung 69
LD LB14235  ; oil supply finish
MOV(021) #0 LD213  ; memory count
; rung 70: P14 END MOTION
LD LB1791  ; P14  Case1 End
OR LB1792  ; P14  Case2 End
OR LB1793  ; P14  Case3 End
OR LB1794  ; P14  Case4 End
OR LB1795  ; P14  Case5 End
OUT LB1799  ; P14 AutoCycleEnd

### Section Device_Output

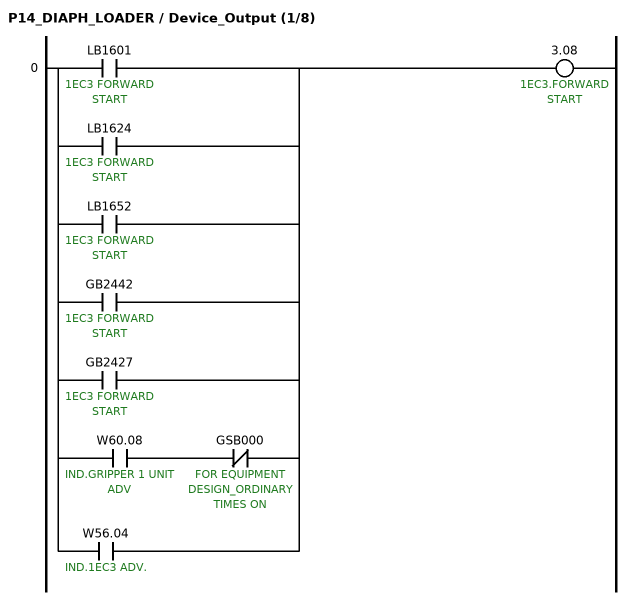
; rung 0
LD LB1601  ; 1EC3 FORWARD START
OR LB1624  ; 1EC3 FORWARD START
OR LB1652  ; 1EC3 FORWARD START
OR GB2442  ; 1EC3 FORWARD START
OR GB2427  ; 1EC3 FORWARD START
LD W60.08  ; IND.GRIPPER 1 UNIT ADV
ANDNOT GSB000  ; FOR EQUIPMENT DESIGN_ORDINARY TIMES ON
ORLD
OR W56.04  ; IND.1EC3 ADV.
OUT 3.08  ; 1EC3.FORWARD START

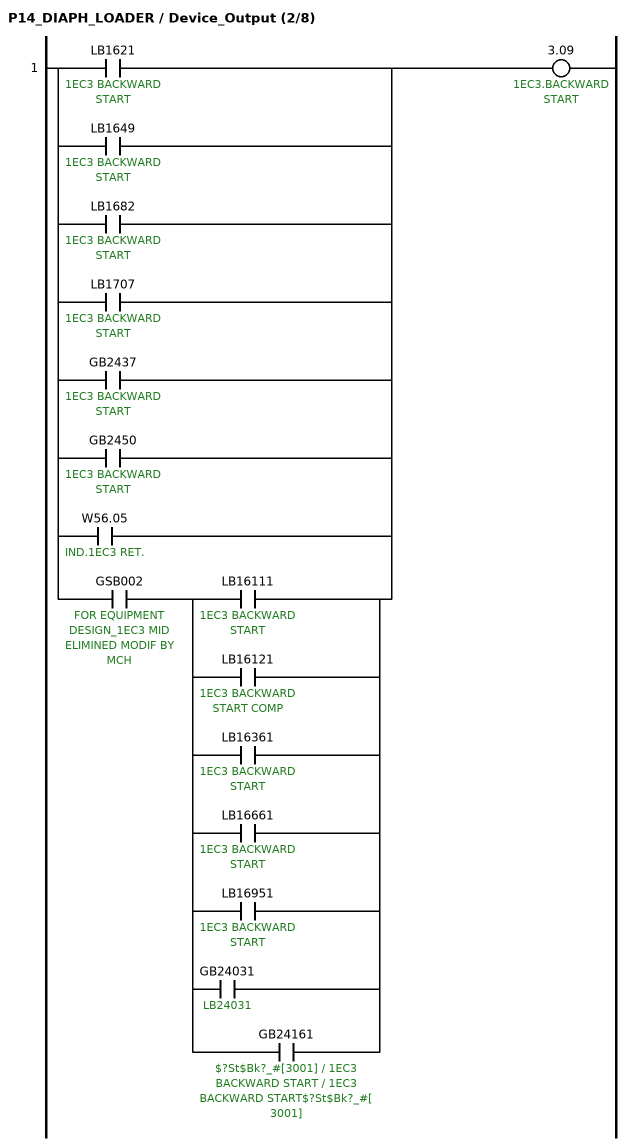
; rung 1
LD LB1621  ; 1EC3 BACKWARD START
OR LB1649  ; 1EC3 BACKWARD START
OR LB1682  ; 1EC3 BACKWARD START
OR LB1707  ; 1EC3 BACKWARD START
OR GB2437  ; 1EC3 BACKWARD START
OR GB2450  ; 1EC3 BACKWARD START
OR W56.05  ; IND.1EC3 RET.
LD GSB002  ; FOR EQUIPMENT DESIGN_1EC3 MID ELIMINED MODIF BY MCH
LD LB16111  ; 1EC3 BACKWARD START
OR LB16121  ; 1EC3 BACKWARD START COMP
OR LB16361  ; 1EC3 BACKWARD START
OR LB16661  ; 1EC3 BACKWARD START
OR LB16951  ; 1EC3 BACKWARD START
OR GB24031  ; LB24031
OR GB24161  ; $?St$Bk?_#[3001] / 1EC3 BACKWARD START / 1EC3 BACKWARD START$?St$Bk?_#[3001]
ANDLD
ORLD
OUT 3.09  ; 1EC3.BACKWARD START

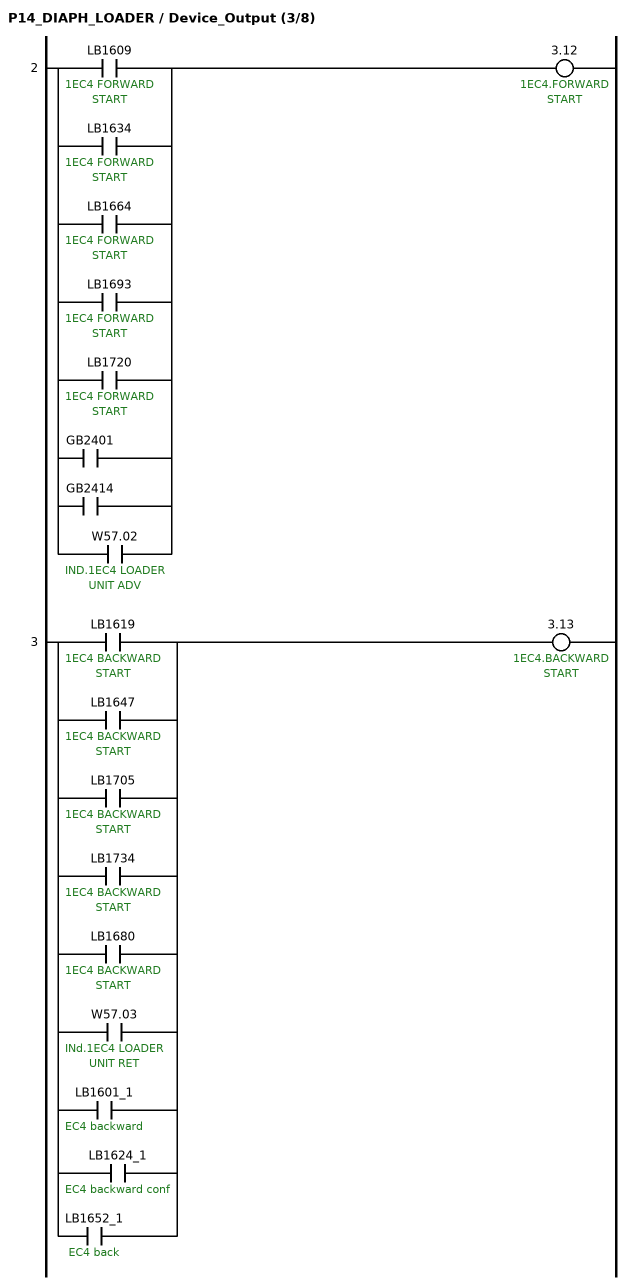
; rung 2
LD LB1609  ; 1EC4 FORWARD START
OR LB1634  ; 1EC4 FORWARD START
OR LB1664  ; 1EC4 FORWARD START
OR LB1693  ; 1EC4 FORWARD START
OR LB1720  ; 1EC4 FORWARD START
OR GB2401
OR GB2414
OR W57.02  ; IND.1EC4 LOADER UNIT ADV
OUT 3.12  ; 1EC4.FORWARD START
; rung 3
LD LB1619  ; 1EC4 BACKWARD START
OR LB1647  ; 1EC4 BACKWARD START
OR LB1705  ; 1EC4 BACKWARD START
OR LB1734  ; 1EC4 BACKWARD START
OR LB1680  ; 1EC4 BACKWARD START
OR W57.03  ; INd.1EC4 LOADER UNIT RET
OR LB1601_1  ; EC4 backward
OR LB1624_1  ; EC4 backward conf
OR LB1652_1  ; EC4 back
OUT 3.13  ; 1EC4.BACKWARD START

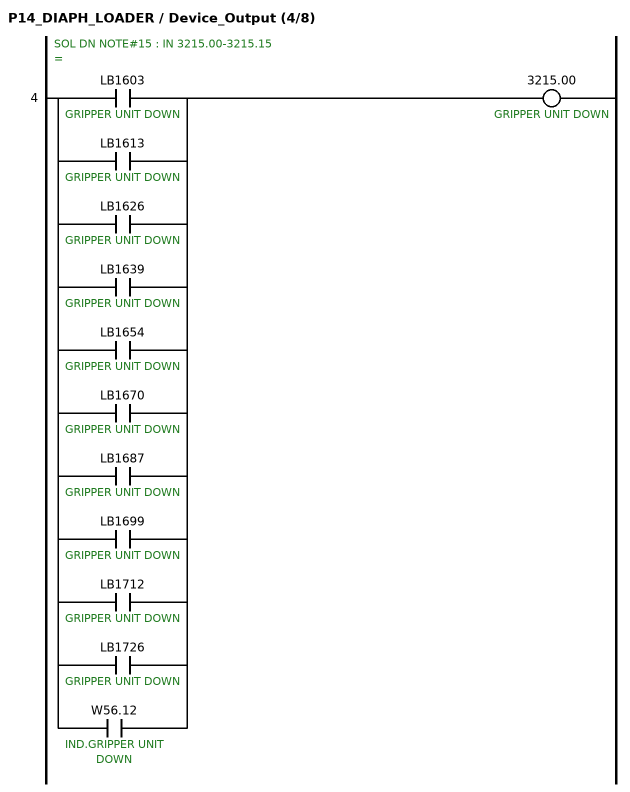
; rung 4: SOL DN NOTE#15 : IN 3215.00-3215.15 / =
LD LB1603  ; GRIPPER UNIT DOWN
OR LB1613  ; GRIPPER UNIT DOWN
OR LB1626  ; GRIPPER UNIT DOWN
OR LB1639  ; GRIPPER UNIT DOWN
OR LB1654  ; GRIPPER UNIT DOWN
OR LB1670  ; GRIPPER UNIT DOWN
OR LB1687  ; GRIPPER UNIT DOWN
OR LB1699  ; GRIPPER UNIT DOWN
OR LB1712  ; GRIPPER UNIT DOWN
OR LB1726  ; GRIPPER UNIT DOWN
OR W56.12  ; IND.GRIPPER UNIT DOWN
OUT 3215.00  ; GRIPPER UNIT DOWN

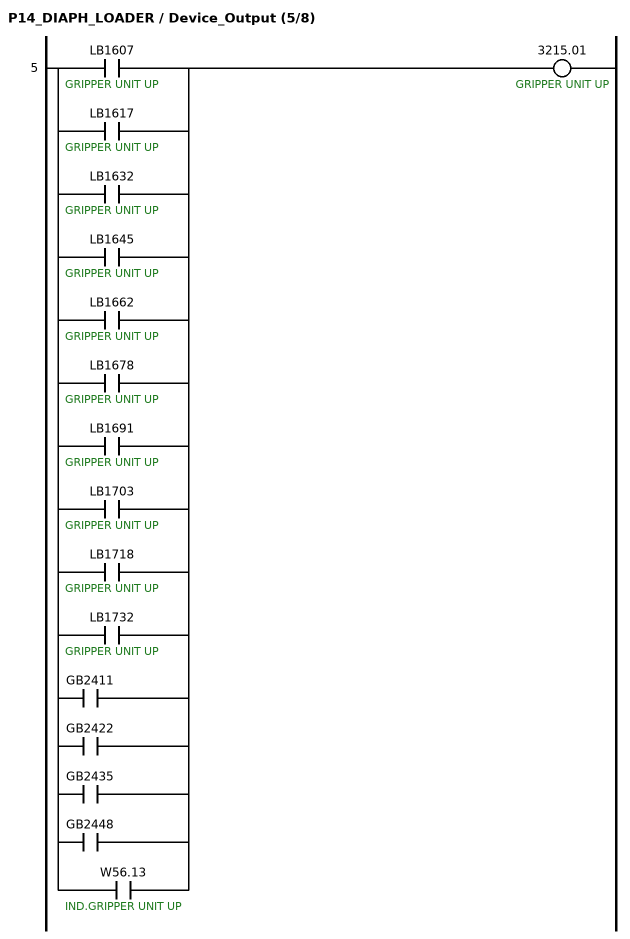
; rung 5
LD LB1607  ; GRIPPER UNIT UP
OR LB1617  ; GRIPPER UNIT UP
OR LB1632  ; GRIPPER UNIT UP
OR LB1645  ; GRIPPER UNIT UP
OR LB1662  ; GRIPPER UNIT UP  // take out all
OR LB1678  ; GRIPPER UNIT UP  // take in all
OR LB1691  ; GRIPPER UNIT UP
OR LB1703  ; GRIPPER UNIT UP
OR LB1718  ; GRIPPER UNIT UP
OR LB1732  ; GRIPPER UNIT UP
OR GB2411
OR GB2422
OR GB2435
OR GB2448
OR W56.13  ; IND.GRIPPER UNIT UP
OUT 3215.01  ; GRIPPER UNIT UP

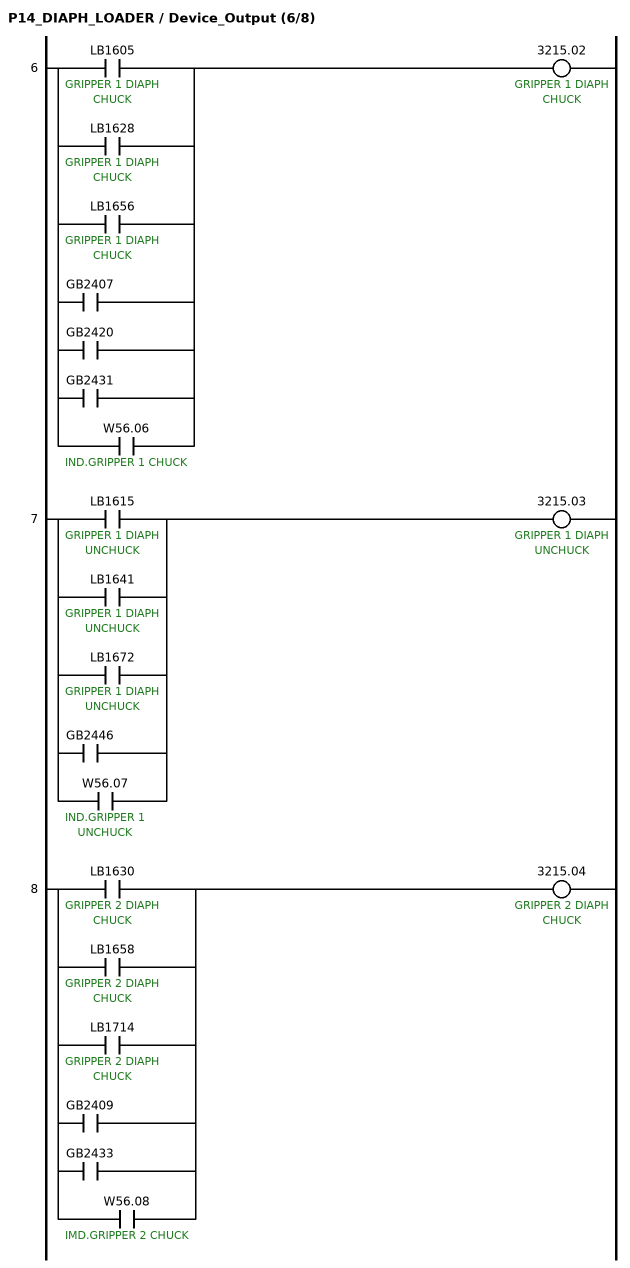
; rung 6
LD LB1605  ; GRIPPER 1 DIAPH CHUCK
OR LB1628  ; GRIPPER 1 DIAPH CHUCK
OR LB1656  ; GRIPPER 1 DIAPH CHUCK
OR GB2407
OR GB2420
OR GB2431
OR W56.06  ; IND.GRIPPER 1 CHUCK
OUT 3215.02  ; GRIPPER 1 DIAPH CHUCK
; rung 7
LD LB1615  ; GRIPPER 1 DIAPH UNCHUCK
OR LB1641  ; GRIPPER 1 DIAPH UNCHUCK
OR LB1672  ; GRIPPER 1 DIAPH UNCHUCK
OR GB2446
OR W56.07  ; IND.GRIPPER 1 UNCHUCK
OUT 3215.03  ; GRIPPER 1 DIAPH UNCHUCK
; rung 8
LD LB1630  ; GRIPPER 2 DIAPH CHUCK
OR LB1658  ; GRIPPER 2 DIAPH CHUCK
OR LB1714  ; GRIPPER 2 DIAPH CHUCK
OR GB2409
OR GB2433
OR W56.08  ; IMD.GRIPPER 2 CHUCK
OUT 3215.04  ; GRIPPER 2 DIAPH CHUCK

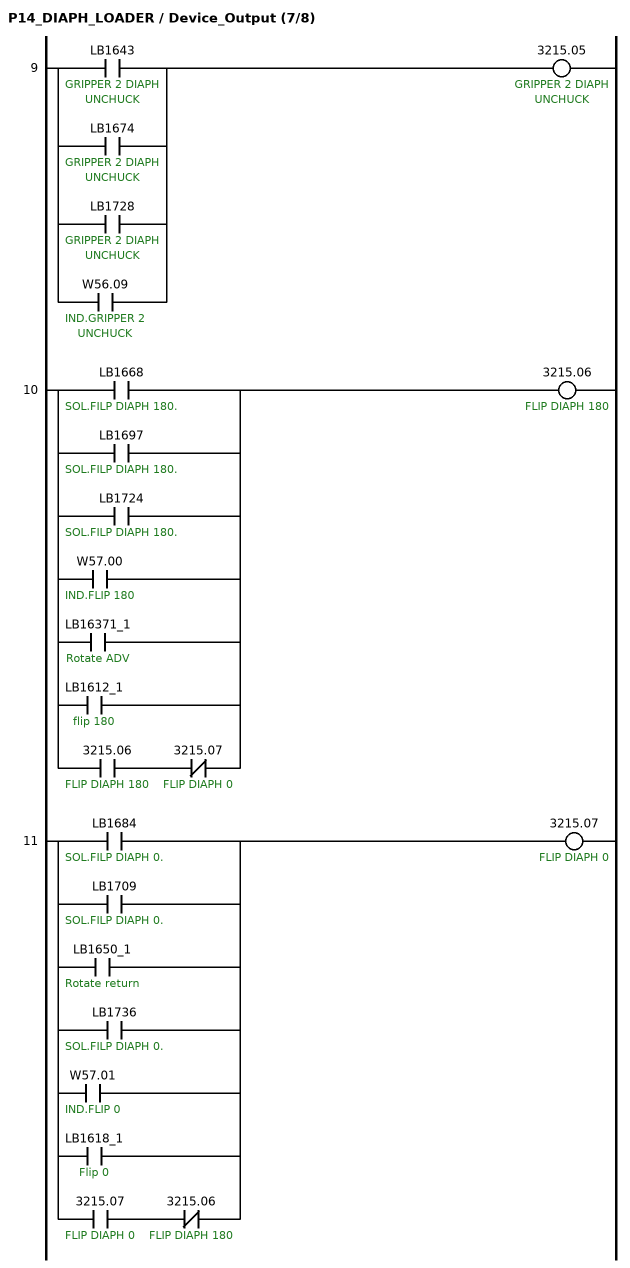
; rung 9
LD LB1643  ; GRIPPER 2 DIAPH UNCHUCK
OR LB1674  ; GRIPPER 2 DIAPH UNCHUCK
OR LB1728  ; GRIPPER 2 DIAPH UNCHUCK
OR W56.09  ; IND.GRIPPER 2 UNCHUCK
OUT 3215.05  ; GRIPPER 2 DIAPH UNCHUCK
; rung 10
LD LB1668  ; SOL.FILP DIAPH 180.
OR LB1697  ; SOL.FILP DIAPH 180.
OR LB1724  ; SOL.FILP DIAPH 180.
OR W57.00  ; IND.FLIP 180
OR LB16371_1  ; Rotate ADV
OR LB1612_1  ; flip 180
LD 3215.06  ; FLIP DIAPH 180
ANDNOT 3215.07  ; FLIP DIAPH 0
ORLD
OUT 3215.06  ; FLIP DIAPH 180
; rung 11
LD LB1684  ; SOL.FILP DIAPH 0.
OR LB1709  ; SOL.FILP DIAPH 0.
OR LB1650_1  ; Rotate return
OR LB1736  ; SOL.FILP DIAPH 0.
OR W57.01  ; IND.FLIP 0
OR LB1618_1  ; Flip 0
LD 3215.07  ; FLIP DIAPH 0
ANDNOT 3215.06  ; FLIP DIAPH 180
ORLD
OUT 3215.07  ; FLIP DIAPH 0

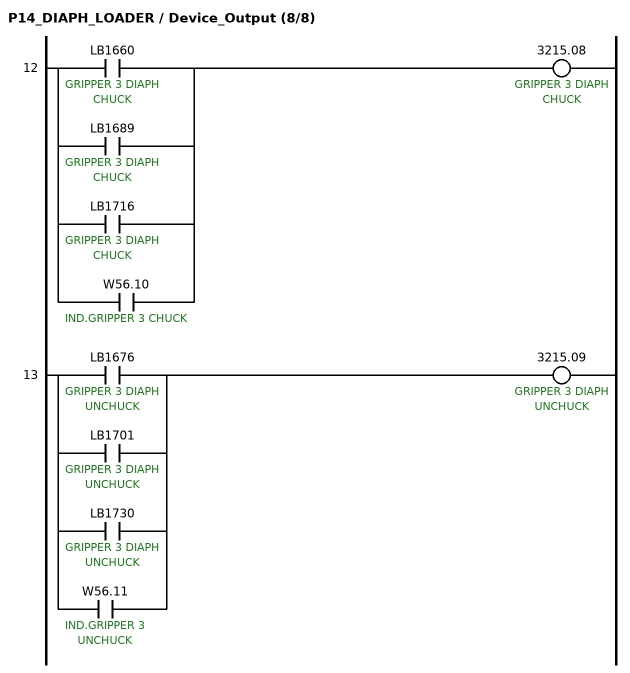
; rung 12
LD LB1660  ; GRIPPER 3 DIAPH CHUCK
OR LB1689  ; GRIPPER 3 DIAPH CHUCK
OR LB1716  ; GRIPPER 3 DIAPH CHUCK
OR W56.10  ; IND.GRIPPER 3 CHUCK
OUT 3215.08  ; GRIPPER 3 DIAPH CHUCK
; rung 13
LD LB1676  ; GRIPPER 3 DIAPH UNCHUCK
OR LB1701  ; GRIPPER 3 DIAPH UNCHUCK
OR LB1730  ; GRIPPER 3 DIAPH UNCHUCK
OR W56.11  ; IND.GRIPPER 3 UNCHUCK
OUT 3215.09  ; GRIPPER 3 DIAPH UNCHUCK

### Section Station_Out

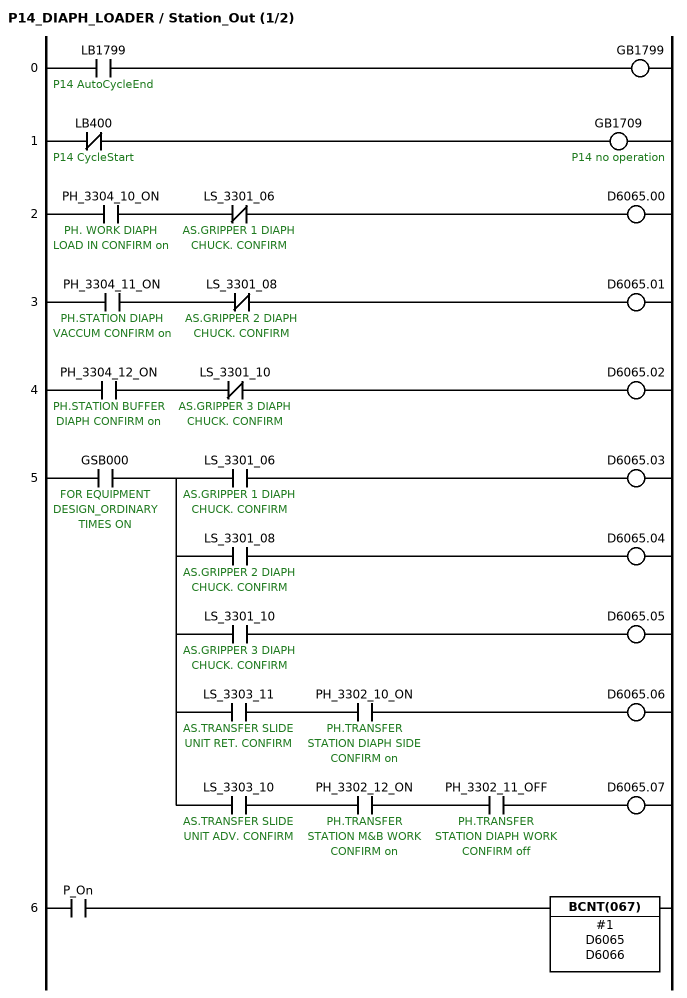
; rung 0
LD LB1799  ; P14 AutoCycleEnd
OUT GB1799
; rung 1
LDNOT LB400  ; P14 CycleStart
OUT GB1709  ; P14 no operation
; rung 2
LD PH_3304_10_ON  ; PH. WORK DIAPH LOAD IN CONFIRM on
ANDNOT LS_3301_06  ; AS.GRIPPER 1 DIAPH CHUCK. CONFIRM
OUT D6065.00
; rung 3
LD PH_3304_11_ON  ; PH.STATION DIAPH VACCUM CONFIRM on
ANDNOT LS_3301_08  ; AS.GRIPPER 2 DIAPH CHUCK. CONFIRM
OUT D6065.01
; rung 4
LD PH_3304_12_ON  ; PH.STATION BUFFER DIAPH CONFIRM on
ANDNOT LS_3301_10  ; AS.GRIPPER 3 DIAPH CHUCK. CONFIRM
OUT D6065.02
; rung 5
LD GSB000  ; FOR EQUIPMENT DESIGN_ORDINARY TIMES ON
OUT TR0
AND LS_3301_06  ; AS.GRIPPER 1 DIAPH CHUCK. CONFIRM
OUT D6065.03
LD TR0
AND LS_3301_08  ; AS.GRIPPER 2 DIAPH CHUCK. CONFIRM
OUT D6065.04
LD TR0
AND LS_3301_10  ; AS.GRIPPER 3 DIAPH CHUCK. CONFIRM
OUT D6065.05
LD TR0
AND LS_3303_11  ; AS.TRANSFER SLIDE UNIT RET. CONFIRM
AND PH_3302_10_ON  ; PH.TRANSFER STATION DIAPH SIDE CONFIRM on
OUT D6065.06
LD TR0
AND LS_3303_10  ; AS.TRANSFER SLIDE UNIT ADV. CONFIRM
AND PH_3302_12_ON  ; PH.TRANSFER STATION M&B WORK CONFIRM on
AND PH_3302_11_OFF  ; PH.TRANSFER STATION DIAPH WORK CONFIRM off
OUT D6065.07
; rung 6
LD P_On
BCNT(067) #1 D6065 D6066

